LIN {X 0,Y 365.471,Z 705.441,A -85,B 0,C 180,E1 17669.142,E2 17669.142} C_VEL
LIN {X 0,Y 364.079,Z 703.275,A -85,B 0,C 180,E1 17668.635,E2 17668.635} C_VEL
LIN {X 0,Y 360.885,Z 700.431,A -85,B 0,C 180,E1 17667.516,E2 17667.516} C_VEL
LIN {X 0,Y 359.152,Z 697.27,A -85,B 0,C 180,E1 17666.808,E2 17666.808} C_VEL
LIN {X 0,Y 355.819,Z 694.962,A -85,B 0,C 180,E1 17665.553,E2 17665.553} C_VEL
LIN {X 0,Y 354.085,Z 691.734,A -85,B 0,C 180,E1 17664.704,E2 17664.704} C_VEL
LIN {X 0,Y 353.877,Z 690.724,A -85,B 0,C 180,E1 17664.135,E2 17664.135} C_VEL
LIN {X 0,Y 353.869,Z 690.629,A -85,B 0,C 180,E1 17659.992,E2 17659.992} C_VEL
LIN {X 0,Y 353.869,Z 690.628,A -85,B 0,C 180,E1 17655.739,E2 17655.739} C_VEL
LIN {X 0,Y 353.867,Z 690.628,A -85,B 0,C 180,E1 17651.573,E2 17651.573} C_VEL
LIN {X 0,Y 353.866,Z 690.63,A -85,B 0,C 180,E1 17647.374,E2 17647.374} C_VEL
LIN {X 0,Y 353.864,Z 690.635,A -85,B 0,C 180,E1 17643.078,E2 17643.078} C_VEL
LIN {X 0,Y 353.868,Z 690.646,A -85,B 0,C 180,E1 17638.867,E2 17638.867} C_VEL
LIN {X 0,Y 353.866,Z 690.656,A -85,B 0,C 180,E1 17634.65,E2 17634.65} C_VEL
LIN {X 0,Y 353.865,Z 690.656,A -85,B 0,C 180,E1 17630.404,E2 17630.404} C_VEL
LIN {X 0,Y 353.855,Z 690.604,A -85,B 0,C 180,E1 17626.103,E2 17626.103} C_VEL
LIN {X 0,Y 353.86,Z 690.613,A -85,B 0,C 180,E1 17622.062,E2 17622.062} C_VEL
LIN {X 0,Y 353.929,Z 691.075,A -85,B 0,C 180,E1 17620.528,E2 17620.528} C_VEL
LIN {X 0,Y 355.457,Z 694.509,A -85,B 0,C 180,E1 17619.242,E2 17619.242} C_VEL
LIN {X 0,Y 357.098,Z 696.566,A -85,B 0,C 180,E1 17618.31,E2 17618.31} C_VEL
LIN {X 0,Y 358.976,Z 700.206,A -85,B 0,C 180,E1 17617.049,E2 17617.049} C_VEL
LIN {X 0,Y 360.256,Z 702.129,A -85,B 0,C 180,E1 17616.328,E2 17616.328} C_VEL
LIN {X 0,Y 363.242,Z 707.517,A -85,B 0,C 180,E1 17614.571,E2 17614.571} C_VEL
LIN {X 0,Y 366.016,Z 712.562,A -85,B 0,C 180,E1 17613.034,E2 17613.034} C_VEL
LIN {X 0,Y 368.872,Z 717.077,A -85,B 0,C 180,E1 17611.859,E2 17611.859} C_VEL
LIN {X 0,Y 376.233,Z 727.791,A -85,B 0,C 180,E1 17609.541,E2 17609.541} C_VEL
LIN {X 0,Y 383.594,Z 738.851,A -85,B 0,C 180,E1 17607.436,E2 17607.436} C_VEL
LIN {X 0,Y 393.463,Z 754.803,A -85,B 0,C 180,E1 17604.86,E2 17604.86} C_VEL
LIN {X 0,Y 403.331,Z 772.096,A -85,B 0,C 180,E1 17602.512,E2 17602.512} C_VEL
LIN {X 0,Y 407.131,Z 779.707,A -85,B 0,C 180,E1 17601.643,E2 17601.643} C_VEL
LIN {X 0,Y 409.573,Z 806.484,A -85,B 0,C 180,E1 17600.521,E2 17600.521} C_VEL
LIN {X 0,Y 399.986,Z 1030.209,A -85,B 0,C 180,E1 17596.253,E2 17596.253} C_VEL
LIN {X 0,Y 398.316,Z 1052.933,A -85,B 0,C 180,E1 17595.707,E2 17595.707} C_VEL
LIN {X 0,Y 395.489,Z 1075.063,A -85,B 0,C 180,E1 17594.972,E2 17594.972} C_VEL
LIN {X 0,Y 391.945,Z 1096.948,A -85,B 0,C 180,E1 17593.997,E2 17593.997} C_VEL
LIN {X 0,Y 388.182,Z 1117.13,A -85,B 0,C 180,E1 17592.842,E2 17592.842} C_VEL
LIN {X 0,Y 383.951,Z 1137.009,A -85,B 0,C 180,E1 17591.409,E2 17591.409} C_VEL
LIN {X 0,Y 379.354,Z 1157.251,A -85,B 0,C 180,E1 17589.629,E2 17589.629} C_VEL
LIN {X 0,Y 374.862,Z 1176.045,A -85,B 0,C 180,E1 17587.646,E2 17587.646} C_VEL
LIN {X 0,Y 370.47,Z 1193.714,A -85,B 0,C 180,E1 17585.407,E2 17585.407} C_VEL
LIN {X 0,Y 366.21,Z 1211.069,A -85,B 0,C 180,E1 17582.807,E2 17582.807} C_VEL
LIN {X 0,Y 362.588,Z 1226.357,A -85,B 0,C 180,E1 17580.123,E2 17580.123} C_VEL
LIN {X 0,Y 359.384,Z 1240.715,A -85,B 0,C 180,E1 17577.146,E2 17577.146} C_VEL
LIN {X 0,Y 356.818,Z 1253.684,A -85,B 0,C 180,E1 17573.973,E2 17573.973} C_VEL
LIN {X 0,Y 354.911,Z 1265.27,A -85,B 0,C 180,E1 17570.618,E2 17570.618} C_VEL
LIN {X 0,Y 353.685,Z 1274.869,A -85,B 0,C 180,E1 17567.267,E2 17567.267} C_VEL
LIN {X 0,Y 353.03,Z 1282.602,A -85,B 0,C 180,E1 17563.93,E2 17563.93} C_VEL
LIN {X 0,Y 352.775,Z 1288.725,A -85,B 0,C 180,E1 17560.616,E2 17560.616} C_VEL
LIN {X 0,Y 352.788,Z 1293.069,A -85,B 0,C 180,E1 17557.327,E2 17557.327} C_VEL
LIN {X 0,Y 352.885,Z 1295.906,A -85,B 0,C 180,E1 17554.062,E2 17554.062} C_VEL
LIN {X 0,Y 352.961,Z 1297.035,A -85,B 0,C 180,E1 17550.974,E2 17550.974} C_VEL
LIN {X 0,Y 352.934,Z 1296.834,A -85,B 0,C 180,E1 17547.889,E2 17547.889} C_VEL
LIN {X 0,Y 352.868,Z 1295.066,A -85,B 0,C 180,E1 17544.798,E2 17544.798} C_VEL
LIN {X 0,Y 352.757,Z 1291.955,A -85,B 0,C 180,E1 17541.689,E2 17541.689} C_VEL
LIN {X 0,Y 352.832,Z 1287.019,A -85,B 0,C 180,E1 17538.393,E2 17538.393} C_VEL
LIN {X 0,Y 353.168,Z 1280.523,A -85,B 0,C 180,E1 17535.071,E2 17535.071} C_VEL
LIN {X 0,Y 353.99,Z 1272.151,A -85,B 0,C 180,E1 17531.729,E2 17531.729} C_VEL
LIN {X 0,Y 355.501,Z 1261.428,A -85,B 0,C 180,E1 17528.208,E2 17528.208} C_VEL
LIN {X 0,Y 357.626,Z 1249.512,A -85,B 0,C 180,E1 17524.937,E2 17524.937} C_VEL
LIN {X 0,Y 360.374,Z 1236.146,A -85,B 0,C 180,E1 17521.859,E2 17521.859} C_VEL
LIN {X 0,Y 363.819,Z 1220.969,A -85,B 0,C 180,E1 17518.892,E2 17518.892} C_VEL
LIN {X 0,Y 367.828,Z 1204.365,A -85,B 0,C 180,E1 17516.136,E2 17516.136} C_VEL
LIN {X 0,Y 372.136,Z 1187.097,A -85,B 0,C 180,E1 17513.71,E2 17513.71} C_VEL
LIN {X 0,Y 376.533,Z 1168.91,A -85,B 0,C 180,E1 17511.568,E2 17511.568} C_VEL
LIN {X 0,Y 381.215,Z 1149.171,A -85,B 0,C 180,E1 17509.623,E2 17509.623} C_VEL
LIN {X 0,Y 385.614,Z 1129.483,A -85,B 0,C 180,E1 17508.014,E2 17508.014} C_VEL
LIN {X 0,Y 389.739,Z 1108.779,A -85,B 0,C 180,E1 17506.655,E2 17506.655} C_VEL
LIN {X 0,Y 393.552,Z 1087.165,A -85,B 0,C 180,E1 17505.535,E2 17505.535} C_VEL
LIN {X 0,Y 396.831,Z 1065.352,A -85,B 0,C 180,E1 17504.682,E2 17504.682} C_VEL
LIN {X 0,Y 399.152,Z 1042.966,A -85,B 0,C 180,E1 17504.036,E2 17504.036} C_VEL
LIN {X 0,Y 400.876,Z 1008.481,A -85,B 0,C 180,E1 17503.333,E2 17503.333} C_VEL
LIN {X 0,Y 409.544,Z 804.991,A -85,B 0,C 180,E1 17499.449,E2 17499.449} C_VEL
LIN {X 0,Y 406.876,Z 778.87,A -85,B 0,C 180,E1 17498.307,E2 17498.307} C_VEL
LIN {X 0,Y 397.759,Z 762.191,A -85,B 0,C 180,E1 17496.208,E2 17496.208} C_VEL
LIN {X 0,Y 387.89,Z 745.698,A -85,B 0,C 180,E1 17493.744,E2 17493.744} C_VEL
LIN {X 0,Y 378.905,Z 731.771,A -85,B 0,C 180,E1 17491.277,E2 17491.277} C_VEL
LIN {X 0,Y 373.111,Z 723.252,A -85,B 0,C 180,E1 17489.543,E2 17489.543} C_VEL
LIN {X 0,Y 367.159,Z 714.598,A -85,B 0,C 180,E1 17487.577,E2 17487.577} C_VEL
LIN {X 0,Y 364.532,Z 709.935,A -85,B 0,C 180,E1 17486.206,E2 17486.206} C_VEL
LIN {X 0,Y 362.094,Z 705.482,A -85,B 0,C 180,E1 17484.817,E2 17484.817} C_VEL
LIN {X 0,Y 359.499,Z 700.812,A -85,B 0,C 180,E1 17483.262,E2 17483.262} C_VEL
LIN {X 0,Y 357.408,Z 697.484,A -85,B 0,C 180,E1 17482.016,E2 17482.016} C_VEL
LIN {X 0,Y 356.62,Z 695.787,A -85,B 0,C 180,E1 17481.44,E2 17481.44} C_VEL
LIN {X 0,Y 354.291,Z 692.379,A -85,B 0,C 180,E1 17479.992,E2 17479.992} C_VEL
LIN {X 0,Y 353.876,Z 690.761,A -85,B 0,C 180,E1 17479.323,E2 17479.323} C_VEL
LIN {X 0,Y 353.859,Z 690.626,A -85,B 0,C 180,E1 17475.067,E2 17475.067} C_VEL
LIN {X 0,Y 353.858,Z 690.634,A -85,B 0,C 180,E1 17470.748,E2 17470.748} C_VEL
LIN {X 0,Y 353.86,Z 690.635,A -85,B 0,C 180,E1 17466.489,E2 17466.489} C_VEL
LIN {X 0,Y 353.858,Z 690.63,A -85,B 0,C 180,E1 17462.267,E2 17462.267} C_VEL
LIN {X 0,Y 353.862,Z 690.627,A -85,B 0,C 180,E1 17458.219,E2 17458.219} C_VEL
LIN {X 0,Y 353.866,Z 690.63,A -85,B 0,C 180,E1 17453.999,E2 17453.999} C_VEL
LIN {X 0,Y 353.87,Z 690.639,A -85,B 0,C 180,E1 17449.911,E2 17449.911} C_VEL
LIN {X 0,Y 353.877,Z 690.644,A -85,B 0,C 180,E1 17445.603,E2 17445.603} C_VEL
LIN {X 0,Y 353.872,Z 690.647,A -85,B 0,C 180,E1 17441.38,E2 17441.38} C_VEL
LIN {X 0,Y 353.873,Z 690.644,A -85,B 0,C 180,E1 17437.084,E2 17437.084} C_VEL
LIN {X 0,Y 353.924,Z 691,A -85,B 0,C 180,E1 17435.456,E2 17435.456} C_VEL
LIN {X 0,Y 354.424,Z 692.729,A -85,B 0,C 180,E1 17434.91,E2 17434.91} C_VEL
LIN {X 0,Y 356.441,Z 695.597,A -85,B 0,C 180,E1 17434.049,E2 17434.049} C_VEL
LIN {X 0,Y 359.358,Z 697.669,A -85,B 0,C 180,E1 17432.963,E2 17432.963} C_VEL
LIN {X 0,Y 361.561,Z 701.257,A -85,B 0,C 180,E1 17432.092,E2 17432.092} C_VEL
LIN {X 0,Y 364.587,Z 703.891,A -85,B 0,C 180,E1 17431.05,E2 17431.05} C_VEL
LIN {X 0,Y 367.355,Z 707.815,A -85,B 0,C 180,E1 17430.081,E2 17430.081} C_VEL
LIN {X 0,Y 369.554,Z 709.947,A -85,B 0,C 180,E1 17429.381,E2 17429.381} C_VEL
LIN {X 0,Y 372.952,Z 714.372,A -85,B 0,C 180,E1 17428.3,E2 17428.3} C_VEL
LIN {X 0,Y 374.652,Z 716.424,A -85,B 0,C 180,E1 17427.786,E2 17427.786} C_VEL
LIN {X 0,Y 379.564,Z 722.657,A -85,B 0,C 180,E1 17426.354,E2 17426.354} C_VEL
LIN {X 0,Y 386.577,Z 731.681,A -85,B 0,C 180,E1 17424.458,E2 17424.458} C_VEL
LIN {X 0,Y 397.204,Z 746.475,A -85,B 0,C 180,E1 17421.831,E2 17421.831} C_VEL
LIN {X 0,Y 408.148,Z 762.945,A -85,B 0,C 180,E1 17419.381,E2 17419.381} C_VEL
LIN {X 0,Y 409.812,Z 765.853,A -85,B 0,C 180,E1 17419.02,E2 17419.02} C_VEL
LIN {X 0,Y 402.072,Z 938.592,A -85,B 0,C 180,E1 17415.686,E2 17415.686} C_VEL
LIN {X 0,Y 400.524,Z 960.749,A -85,B 0,C 180,E1 17415.004,E2 17415.004} C_VEL
LIN {X 0,Y 398.362,Z 981.552,A -85,B 0,C 180,E1 17414.123,E2 17414.123} C_VEL
LIN {X 0,Y 395.581,Z 1001.394,A -85,B 0,C 180,E1 17413.033,E2 17413.033} C_VEL
LIN {X 0,Y 392.215,Z 1020.769,A -85,B 0,C 180,E1 17411.708,E2 17411.708} C_VEL
LIN {X 0,Y 388.601,Z 1038.719,A -85,B 0,C 180,E1 17410.225,E2 17410.225} C_VEL
LIN {X 0,Y 384.411,Z 1056.584,A -85,B 0,C 180,E1 17408.435,E2 17408.435} C_VEL
LIN {X 0,Y 379.966,Z 1073.805,A -85,B 0,C 180,E1 17406.368,E2 17406.368} C_VEL
LIN {X 0,Y 375.604,Z 1089.572,A -85,B 0,C 180,E1 17404.118,E2 17404.118} C_VEL
LIN {X 0,Y 371.339,Z 1103.939,A -85,B 0,C 180,E1 17401.671,E2 17401.671} C_VEL
LIN {X 0,Y 367.297,Z 1117.2,A -85,B 0,C 180,E1 17398.982,E2 17398.982} C_VEL
LIN {X 0,Y 363.656,Z 1129.181,A -85,B 0,C 180,E1 17396.097,E2 17396.097} C_VEL
LIN {X 0,Y 360.477,Z 1139.749,A -85,B 0,C 180,E1 17393.022,E2 17393.022} C_VEL
LIN {X 0,Y 357.859,Z 1148.935,A -85,B 0,C 180,E1 17389.759,E2 17389.759} C_VEL
LIN {X 0,Y 355.866,Z 1156.767,A -85,B 0,C 180,E1 17386.317,E2 17386.317} C_VEL
LIN {X 0,Y 354.504,Z 1162.89,A -85,B 0,C 180,E1 17382.874,E2 17382.874} C_VEL
LIN {X 0,Y 353.689,Z 1167.41,A -85,B 0,C 180,E1 17379.388,E2 17379.388} C_VEL
LIN {X 0,Y 353.21,Z 1170.657,A -85,B 0,C 180,E1 17375.686,E2 17375.686} C_VEL
LIN {X 0,Y 353.051,Z 1172.217,A -85,B 0,C 180,E1 17372.4,E2 17372.4} C_VEL
LIN {X 0,Y 352.043,Z 1172.727,A -85,B 0,C 180,E1 17371.152,E2 17371.152} C_VEL
LIN {X 0,Y 347.31,Z 1173.512,A -85,B 0,C 180,E1 17368.703,E2 17368.703} C_VEL
LIN {X 0,Y 345.319,Z 1173.487,A -85,B 0,C 180,E1 17367.162,E2 17367.162} C_VEL
LIN {X 0,Y 345.197,Z 1173.339,A -85,B 0,C 180,E1 17366.699,E2 17366.699} C_VEL
LIN {X 0,Y 345.475,Z 1171.37,A -85,B 0,C 180,E1 17363.072,E2 17363.072} C_VEL
LIN {X 0,Y 346.007,Z 1168.136,A -85,B 0,C 180,E1 17359.679,E2 17359.679} C_VEL
LIN {X 0,Y 347.031,Z 1163.092,A -85,B 0,C 180,E1 17355.995,E2 17355.995} C_VEL
LIN {X 0,Y 348.637,Z 1156.696,A -85,B 0,C 180,E1 17352.475,E2 17352.475} C_VEL
LIN {X 0,Y 350.95,Z 1148.496,A -85,B 0,C 180,E1 17348.963,E2 17348.963} C_VEL
LIN {X 0,Y 353.886,Z 1138.82,A -85,B 0,C 180,E1 17345.639,E2 17345.639} C_VEL
LIN {X 0,Y 357.626,Z 1127.14,A -85,B 0,C 180,E1 17342.349,E2 17342.349} C_VEL
LIN {X 0,Y 361.695,Z 1114.634,A -85,B 0,C 180,E1 17339.428,E2 17339.428} C_VEL
LIN {X 0,Y 366.129,Z 1100.591,A -85,B 0,C 180,E1 17336.709,E2 17336.709} C_VEL
LIN {X 0,Y 370.63,Z 1085.712,A -85,B 0,C 180,E1 17334.294,E2 17334.294} C_VEL
LIN {X 0,Y 375.04,Z 1070.375,A -85,B 0,C 180,E1 17332.181,E2 17332.181} C_VEL
LIN {X 0,Y 379.54,Z 1053.085,A -85,B 0,C 180,E1 17330.198,E2 17330.198} C_VEL
LIN {X 0,Y 383.74,Z 1034.99,A -85,B 0,C 180,E1 17328.464,E2 17328.464} C_VEL
LIN {X 0,Y 387.565,Z 1016.262,A -85,B 0,C 180,E1 17326.973,E2 17326.973} C_VEL
LIN {X 0,Y 390.864,Z 996.564,A -85,B 0,C 180,E1 17325.707,E2 17325.707} C_VEL
LIN {X 0,Y 393.661,Z 975.449,A -85,B 0,C 180,E1 17324.633,E2 17324.633} C_VEL
LIN {X 0,Y 395.75,Z 954.159,A -85,B 0,C 180,E1 17323.812,E2 17323.812} C_VEL
LIN {X 0,Y 396.956,Z 933.715,A -85,B 0,C 180,E1 17323.253,E2 17323.253} C_VEL
LIN {X 0,Y 404.544,Z 769.328,A -85,B 0,C 180,E1 17320.063,E2 17320.063} C_VEL
LIN {X 0,Y 393.935,Z 753.113,A -85,B 0,C 180,E1 17317.62,E2 17317.62} C_VEL
LIN {X 0,Y 384.99,Z 740.534,A -85,B 0,C 180,E1 17315.367,E2 17315.367} C_VEL
LIN {X 0,Y 378.062,Z 731.268,A -85,B 0,C 180,E1 17313.465,E2 17313.465} C_VEL
LIN {X 0,Y 374.232,Z 726.376,A -85,B 0,C 180,E1 17312.346,E2 17312.346} C_VEL
LIN {X 0,Y 370.309,Z 721.384,A -85,B 0,C 180,E1 17311.136,E2 17311.136} C_VEL
LIN {X 0,Y 365.999,Z 715.983,A -85,B 0,C 180,E1 17309.725,E2 17309.725} C_VEL
LIN {X 0,Y 362.579,Z 711.859,A -85,B 0,C 180,E1 17308.539,E2 17308.539} C_VEL
LIN {X 0,Y 361.48,Z 710.424,A -85,B 0,C 180,E1 17308.139,E2 17308.139} C_VEL
LIN {X 0,Y 358.283,Z 707.187,A -85,B 0,C 180,E1 17306.968,E2 17306.968} C_VEL
LIN {X 0,Y 356.638,Z 704.578,A -85,B 0,C 180,E1 17306.293,E2 17306.293} C_VEL
LIN {X 0,Y 353.417,Z 701.9,A -85,B 0,C 180,E1 17305.021,E2 17305.021} C_VEL
LIN {X 0,Y 351.252,Z 698.256,A -85,B 0,C 180,E1 17304.02,E2 17304.02} C_VEL
LIN {X 0,Y 347.935,Z 696.011,A -85,B 0,C 180,E1 17302.559,E2 17302.559} C_VEL
LIN {X 0,Y 346.135,Z 692.717,A -85,B 0,C 180,E1 17301.522,E2 17301.522} C_VEL
LIN {X 0,Y 345.941,Z 691.687,A -85,B 0,C 180,E1 17300.824,E2 17300.824} C_VEL
LIN {X 0,Y 345.932,Z 691.618,A -85,B 0,C 180,E1 17296.455,E2 17296.455} C_VEL
LIN {X 0,Y 345.93,Z 691.62,A -85,B 0,C 180,E1 17292.181,E2 17292.181} C_VEL
LIN {X 0,Y 345.938,Z 691.621,A -85,B 0,C 180,E1 17287.808,E2 17287.808} C_VEL
LIN {X 0,Y 345.928,Z 691.629,A -85,B 0,C 180,E1 17283.48,E2 17283.48} C_VEL
LIN {X 0,Y 345.935,Z 691.64,A -85,B 0,C 180,E1 17279.172,E2 17279.172} C_VEL
LIN {X 0,Y 345.931,Z 691.647,A -85,B 0,C 180,E1 17274.86,E2 17274.86} C_VEL
LIN {X 0,Y 345.928,Z 691.638,A -85,B 0,C 180,E1 17270.685,E2 17270.685} C_VEL
LIN {X 0,Y 345.924,Z 691.587,A -85,B 0,C 180,E1 17266.46,E2 17266.46} C_VEL
LIN {X 0,Y 345.978,Z 691.985,A -85,B 0,C 180,E1 17263.32,E2 17263.32} C_VEL
LIN {X 0,Y 347.643,Z 695.648,A -85,B 0,C 180,E1 17261.73,E2 17261.73} C_VEL
LIN {X 0,Y 349.357,Z 697.89,A -85,B 0,C 180,E1 17260.611,E2 17260.611} C_VEL
LIN {X 0,Y 351.358,Z 701.541,A -85,B 0,C 180,E1 17259.163,E2 17259.163} C_VEL
LIN {X 0,Y 352.421,Z 703.029,A -85,B 0,C 180,E1 17258.52,E2 17258.52} C_VEL
LIN {X 0,Y 354.585,Z 706.924,A -85,B 0,C 180,E1 17257.1,E2 17257.1} C_VEL
LIN {X 0,Y 357.639,Z 711.946,A -85,B 0,C 180,E1 17255.471,E2 17255.471} C_VEL
LIN {X 0,Y 365.872,Z 723.456,A -85,B 0,C 180,E1 17252.45,E2 17252.45} C_VEL
LIN {X 0,Y 373.526,Z 734.859,A -85,B 0,C 180,E1 17249.963,E2 17249.963} C_VEL
LIN {X 0,Y 380.424,Z 745.435,A -85,B 0,C 180,E1 17247.933,E2 17247.933} C_VEL
LIN {X 0,Y 390.016,Z 761.232,A -85,B 0,C 180,E1 17245.356,E2 17245.356} C_VEL
LIN {X 0,Y 399.414,Z 777.97,A -85,B 0,C 180,E1 17243.051,E2 17243.051} C_VEL
LIN {X 0,Y 402.235,Z 783.755,A -85,B 0,C 180,E1 17242.381,E2 17242.381} C_VEL
LIN {X 0,Y 404.318,Z 807.97,A -85,B 0,C 180,E1 17241.354,E2 17241.354} C_VEL
LIN {X 0,Y 394.338,Z 1030.205,A -85,B 0,C 180,E1 17237.074,E2 17237.074} C_VEL
LIN {X 0,Y 392.557,Z 1052.868,A -85,B 0,C 180,E1 17236.516,E2 17236.516} C_VEL
LIN {X 0,Y 389.542,Z 1075.287,A -85,B 0,C 180,E1 17235.753,E2 17235.753} C_VEL
LIN {X 0,Y 385.961,Z 1096.296,A -85,B 0,C 180,E1 17234.798,E2 17234.798} C_VEL
LIN {X 0,Y 381.963,Z 1116.754,A -85,B 0,C 180,E1 17233.609,E2 17233.609} C_VEL
LIN {X 0,Y 377.446,Z 1137.037,A -85,B 0,C 180,E1 17232.122,E2 17232.122} C_VEL
LIN {X 0,Y 372.825,Z 1156.344,A -85,B 0,C 180,E1 17230.391,E2 17230.391} C_VEL
LIN {X 0,Y 368.084,Z 1175.208,A -85,B 0,C 180,E1 17228.365,E2 17228.365} C_VEL
LIN {X 0,Y 363.438,Z 1193.028,A -85,B 0,C 180,E1 17226.066,E2 17226.066} C_VEL
LIN {X 0,Y 359.03,Z 1210.026,A -85,B 0,C 180,E1 17223.462,E2 17223.462} C_VEL
LIN {X 0,Y 355.085,Z 1225.698,A -85,B 0,C 180,E1 17220.64,E2 17220.64} C_VEL
LIN {X 0,Y 351.612,Z 1240.558,A -85,B 0,C 180,E1 17217.475,E2 17217.475} C_VEL
LIN {X 0,Y 348.917,Z 1253.462,A -85,B 0,C 180,E1 17214.19,E2 17214.19} C_VEL
LIN {X 0,Y 346.958,Z 1264.821,A -85,B 0,C 180,E1 17210.76,E2 17210.76} C_VEL
LIN {X 0,Y 345.71,Z 1274.303,A -85,B 0,C 180,E1 17207.331,E2 17207.331} C_VEL
LIN {X 0,Y 345.065,Z 1281.866,A -85,B 0,C 180,E1 17203.907,E2 17203.907} C_VEL
LIN {X 0,Y 344.845,Z 1288.021,A -85,B 0,C 180,E1 17200.356,E2 17200.356} C_VEL
LIN {X 0,Y 344.882,Z 1292.027,A -85,B 0,C 180,E1 17197.161,E2 17197.161} C_VEL
LIN {X 0,Y 345.008,Z 1294.674,A -85,B 0,C 180,E1 17193.822,E2 17193.822} C_VEL
LIN {X 0,Y 345.08,Z 1295.669,A -85,B 0,C 180,E1 17190.83,E2 17190.83} C_VEL
LIN {X 0,Y 345.043,Z 1295.301,A -85,B 0,C 180,E1 17187.509,E2 17187.509} C_VEL
LIN {X 0,Y 344.951,Z 1293.532,A -85,B 0,C 180,E1 17184.511,E2 17184.511} C_VEL
LIN {X 0,Y 344.835,Z 1290.355,A -85,B 0,C 180,E1 17181.328,E2 17181.328} C_VEL
LIN {X 0,Y 344.914,Z 1285.3,A -85,B 0,C 180,E1 17177.953,E2 17177.953} C_VEL
LIN {X 0,Y 345.323,Z 1278.286,A -85,B 0,C 180,E1 17174.379,E2 17174.379} C_VEL
LIN {X 0,Y 346.187,Z 1270.233,A -85,B 0,C 180,E1 17171.127,E2 17171.127} C_VEL
LIN {X 0,Y 347.745,Z 1259.95,A -85,B 0,C 180,E1 17167.696,E2 17167.696} C_VEL
LIN {X 0,Y 349.949,Z 1248.388,A -85,B 0,C 180,E1 17164.442,E2 17164.442} C_VEL
LIN {X 0,Y 352.952,Z 1234.654,A -85,B 0,C 180,E1 17161.212,E2 17161.212} C_VEL
LIN {X 0,Y 356.618,Z 1219.477,A -85,B 0,C 180,E1 17158.191,E2 17158.191} C_VEL
LIN {X 0,Y 360.891,Z 1202.746,A -85,B 0,C 180,E1 17155.37,E2 17155.37} C_VEL
LIN {X 0,Y 365.456,Z 1185.367,A -85,B 0,C 180,E1 17152.897,E2 17152.897} C_VEL
LIN {X 0,Y 370.161,Z 1166.853,A -85,B 0,C 180,E1 17150.699,E2 17150.699} C_VEL
LIN {X 0,Y 375.092,Z 1147.001,A -85,B 0,C 180,E1 17148.738,E2 17148.738} C_VEL
LIN {X 0,Y 379.508,Z 1128.019,A -85,B 0,C 180,E1 17147.179,E2 17147.179} C_VEL
LIN {X 0,Y 383.778,Z 1107.455,A -85,B 0,C 180,E1 17145.821,E2 17145.821} C_VEL
LIN {X 0,Y 387.796,Z 1085.627,A -85,B 0,C 180,E1 17144.688,E2 17144.688} C_VEL
LIN {X 0,Y 391.182,Z 1063.831,A -85,B 0,C 180,E1 17143.835,E2 17143.835} C_VEL
LIN {X 0,Y 393.571,Z 1041.356,A -85,B 0,C 180,E1 17143.183,E2 17143.183} C_VEL
LIN {X 0,Y 395.395,Z 1006,A -85,B 0,C 180,E1 17142.458,E2 17142.458} C_VEL
LIN {X 0,Y 404.287,Z 806.378,A -85,B 0,C 180,E1 17138.613,E2 17138.613} C_VEL
LIN {X 0,Y 401.977,Z 782.959,A -85,B 0,C 180,E1 17137.568,E2 17137.568} C_VEL
LIN {X 0,Y 393.041,Z 766.442,A -85,B 0,C 180,E1 17135.428,E2 17135.428} C_VEL
LIN {X 0,Y 382.85,Z 749.242,A -85,B 0,C 180,E1 17132.769,E2 17132.769} C_VEL
LIN {X 0,Y 374.337,Z 736.079,A -85,B 0,C 180,E1 17130.319,E2 17130.319} C_VEL
LIN {X 0,Y 367.967,Z 726.664,A -85,B 0,C 180,E1 17128.304,E2 17128.304} C_VEL
LIN {X 0,Y 363.794,Z 720.659,A -85,B 0,C 180,E1 17126.879,E2 17126.879} C_VEL
LIN {X 0,Y 357.321,Z 711.598,A -85,B 0,C 180,E1 17124.465,E2 17124.465} C_VEL
LIN {X 0,Y 354.502,Z 706.829,A -85,B 0,C 180,E1 17122.906,E2 17122.906} C_VEL
LIN {X 0,Y 352.349,Z 702.839,A -85,B 0,C 180,E1 17121.473,E2 17121.473} C_VEL
LIN {X 0,Y 349.639,Z 698.685,A -85,B 0,C 180,E1 17119.721,E2 17119.721} C_VEL
LIN {X 0,Y 348.867,Z 696.937,A -85,B 0,C 180,E1 17119.07,E2 17119.07} C_VEL
LIN {X 0,Y 346.498,Z 693.756,A -85,B 0,C 180,E1 17117.463,E2 17117.463} C_VEL
LIN {X 0,Y 345.956,Z 691.853,A -85,B 0,C 180,E1 17116.626,E2 17116.626} C_VEL
LIN {X 0,Y 345.918,Z 691.588,A -85,B 0,C 180,E1 17112.52,E2 17112.52} C_VEL
LIN {X 0,Y 345.923,Z 691.621,A -85,B 0,C 180,E1 17108.309,E2 17108.309} C_VEL
LIN {X 0,Y 345.92,Z 691.629,A -85,B 0,C 180,E1 17104.144,E2 17104.144} C_VEL
LIN {X 0,Y 345.923,Z 691.637,A -85,B 0,C 180,E1 17099.834,E2 17099.834} C_VEL
LIN {X 0,Y 345.922,Z 691.647,A -85,B 0,C 180,E1 17095.524,E2 17095.524} C_VEL
LIN {X 0,Y 345.921,Z 691.641,A -85,B 0,C 180,E1 17091.299,E2 17091.299} C_VEL
LIN {X 0,Y 345.922,Z 691.634,A -85,B 0,C 180,E1 17086.97,E2 17086.97} C_VEL
LIN {X 0,Y 345.923,Z 691.629,A -85,B 0,C 180,E1 17082.679,E2 17082.679} C_VEL
LIN {X 0,Y 345.952,Z 691.793,A -85,B 0,C 180,E1 17078.821,E2 17078.821} C_VEL
LIN {X 0,Y 346.263,Z 693.135,A -85,B 0,C 180,E1 17078.175,E2 17078.175} C_VEL
LIN {X 0,Y 347.944,Z 696.018,A -85,B 0,C 180,E1 17077.272,E2 17077.272} C_VEL
LIN {X 0,Y 351.639,Z 698.72,A -85,B 0,C 180,E1 17075.651,E2 17075.651} C_VEL
LIN {X 0,Y 353.739,Z 702.299,A -85,B 0,C 180,E1 17074.69,E2 17074.69} C_VEL
LIN {X 0,Y 357.083,Z 705.131,A -85,B 0,C 180,E1 17073.384,E2 17073.384} C_VEL
LIN {X 0,Y 359.722,Z 708.944,A -85,B 0,C 180,E1 17072.342,E2 17072.342} C_VEL
LIN {X 0,Y 362.185,Z 711.201,A -85,B 0,C 180,E1 17071.472,E2 17071.472} C_VEL
LIN {X 0,Y 365.461,Z 715.501,A -85,B 0,C 180,E1 17070.317,E2 17070.317} C_VEL
LIN {X 0,Y 367.18,Z 717.401,A -85,B 0,C 180,E1 17069.75,E2 17069.75} C_VEL
LIN {X 0,Y 371.011,Z 722.061,A -85,B 0,C 180,E1 17068.523,E2 17068.523} C_VEL
LIN {X 0,Y 380.126,Z 733.931,A -85,B 0,C 180,E1 17065.835,E2 17065.835} C_VEL
LIN {X 0,Y 390.273,Z 747.832,A -85,B 0,C 180,E1 17063.166,E2 17063.166} C_VEL
LIN {X 0,Y 400.617,Z 763.242,A -85,B 0,C 180,E1 17060.705,E2 17060.705} C_VEL
LIN {X 0,Y 404.549,Z 769.661,A -85,B 0,C 180,E1 17059.821,E2 17059.821} C_VEL
LIN {X 0,Y 396.607,Z 939.648,A -85,B 0,C 180,E1 17056.512,E2 17056.512} C_VEL
LIN {X 0,Y 395.01,Z 961.899,A -85,B 0,C 180,E1 17055.823,E2 17055.823} C_VEL
LIN {X 0,Y 392.855,Z 982.158,A -85,B 0,C 180,E1 17054.965,E2 17054.965} C_VEL
LIN {X 0,Y 390.049,Z 1001.546,A -85,B 0,C 180,E1 17053.899,E2 17053.899} C_VEL
LIN {X 0,Y 386.561,Z 1021.196,A -85,B 0,C 180,E1 17052.56,E2 17052.56} C_VEL
LIN {X 0,Y 382.801,Z 1039.298,A -85,B 0,C 180,E1 17051.063,E2 17051.063} C_VEL
LIN {X 0,Y 378.512,Z 1056.971,A -85,B 0,C 180,E1 17049.287,E2 17049.287} C_VEL
LIN {X 0,Y 373.71,Z 1074.91,A -85,B 0,C 180,E1 17047.127,E2 17047.127} C_VEL
LIN {X 0,Y 369.147,Z 1090.744,A -85,B 0,C 180,E1 17044.845,E2 17044.845} C_VEL
LIN {X 0,Y 364.608,Z 1105.342,A -85,B 0,C 180,E1 17042.326,E2 17042.326} C_VEL
LIN {X 0,Y 360.362,Z 1118.605,A -85,B 0,C 180,E1 17039.595,E2 17039.595} C_VEL
LIN {X 0,Y 356.523,Z 1130.588,A -85,B 0,C 180,E1 17036.66,E2 17036.66} C_VEL
LIN {X 0,Y 353.07,Z 1141.461,A -85,B 0,C 180,E1 17033.431,E2 17033.431} C_VEL
LIN {X 0,Y 350.255,Z 1150.758,A -85,B 0,C 180,E1 17030.032,E2 17030.032} C_VEL
LIN {X 0,Y 348.069,Z 1158.805,A -85,B 0,C 180,E1 17026.35,E2 17026.35} C_VEL
LIN {X 0,Y 346.668,Z 1164.793,A -85,B 0,C 180,E1 17022.831,E2 17022.831} C_VEL
LIN {X 0,Y 345.828,Z 1169.118,A -85,B 0,C 180,E1 17019.317,E2 17019.317} C_VEL
LIN {X 0,Y 345.338,Z 1172.149,A -85,B 0,C 180,E1 17015.649,E2 17015.649} C_VEL
LIN {X 0,Y 345.169,Z 1173.714,A -85,B 0,C 180,E1 17012.158,E2 17012.158} C_VEL
LIN {X 0,Y 345.15,Z 1173.824,A -85,B 0,C 180,E1 17008.672,E2 17008.672} C_VEL
LIN {X 0,Y 345.197,Z 1173.339,A -85,B 0,C 180,E1 17006.699,E2 17006.699} C_VEL
LIN {X 0,Y 344.3,Z 1173.029,A -85,B 0,C 180,E1 17005.419,E2 17005.419} C_VEL
LIN {X 0,Y 338.432,Z 1171.92,A -85,B 0,C 180,E1 17001.889,E2 17001.889} C_VEL
LIN {X 0,Y 337.945,Z 1171.047,A -85,B 0,C 180,E1 17000.863,E2 17000.863} C_VEL
LIN {X 0,Y 338.794,Z 1166.769,A -85,B 0,C 180,E1 16997.213,E2 16997.213} C_VEL
LIN {X 0,Y 340.319,Z 1160.704,A -85,B 0,C 180,E1 16993.442,E2 16993.442} C_VEL
LIN {X 0,Y 342.476,Z 1153.233,A -85,B 0,C 180,E1 16989.849,E2 16989.849} C_VEL
LIN {X 0,Y 345.304,Z 1144.354,A -85,B 0,C 180,E1 16986.448,E2 16986.448} C_VEL
LIN {X 0,Y 348.721,Z 1134.068,A -85,B 0,C 180,E1 16983.247,E2 16983.247} C_VEL
LIN {X 0,Y 352.885,Z 1121.83,A -85,B 0,C 180,E1 16980.089,E2 16980.089} C_VEL
LIN {X 0,Y 357.264,Z 1108.919,A -85,B 0,C 180,E1 16977.308,E2 16977.308} C_VEL
LIN {X 0,Y 361.922,Z 1094.514,A -85,B 0,C 180,E1 16974.734,E2 16974.734} C_VEL
LIN {X 0,Y 366.923,Z 1078.185,A -85,B 0,C 180,E1 16972.285,E2 16972.285} C_VEL
LIN {X 0,Y 371.674,Z 1061.501,A -85,B 0,C 180,E1 16970.191,E2 16970.191} C_VEL
LIN {X 0,Y 376.142,Z 1043.857,A -85,B 0,C 180,E1 16968.354,E2 16968.354} C_VEL
LIN {X 0,Y 380.318,Z 1025.143,A -85,B 0,C 180,E1 16966.739,E2 16966.739} C_VEL
LIN {X 0,Y 383.874,Z 1006.668,A -85,B 0,C 180,E1 16965.418,E2 16965.418} C_VEL
LIN {X 0,Y 386.897,Z 986.887,A -85,B 0,C 180,E1 16964.289,E2 16964.289} C_VEL
LIN {X 0,Y 389.451,Z 965.005,A -85,B 0,C 180,E1 16963.315,E2 16963.315} C_VEL
LIN {X 0,Y 391.142,Z 943.712,A -85,B 0,C 180,E1 16962.617,E2 16962.617} C_VEL
LIN {X 0,Y 393.475,Z 894.086,A -85,B 0,C 180,E1 16961.592,E2 16961.592} C_VEL
LIN {X 0,Y 399.302,Z 773.086,A -85,B 0,C 180,E1 16959.227,E2 16959.227} C_VEL
LIN {X 0,Y 388.852,Z 757.058,A -85,B 0,C 180,E1 16956.715,E2 16956.715} C_VEL
LIN {X 0,Y 379.24,Z 743.486,A -85,B 0,C 180,E1 16954.165,E2 16954.165} C_VEL
LIN {X 0,Y 371.689,Z 733.528,A -85,B 0,C 180,E1 16951.956,E2 16951.956} C_VEL
LIN {X 0,Y 367.378,Z 728.068,A -85,B 0,C 180,E1 16950.594,E2 16950.594} C_VEL
LIN {X 0,Y 363.359,Z 722.964,A -85,B 0,C 180,E1 16949.238,E2 16949.238} C_VEL
LIN {X 0,Y 359.822,Z 718.436,A -85,B 0,C 180,E1 16947.964,E2 16947.964} C_VEL
LIN {X 0,Y 355.714,Z 713.936,A -85,B 0,C 180,E1 16946.412,E2 16946.412} C_VEL
LIN {X 0,Y 354.355,Z 711.94,A -85,B 0,C 180,E1 16945.846,E2 16945.846} C_VEL
LIN {X 0,Y 351.048,Z 708.817,A -85,B 0,C 180,E1 16944.483,E2 16944.483} C_VEL
LIN {X 0,Y 349.251,Z 705.805,A -85,B 0,C 180,E1 16943.629,E2 16943.629} C_VEL
LIN {X 0,Y 346.016,Z 703.383,A -85,B 0,C 180,E1 16942.154,E2 16942.154} C_VEL
LIN {X 0,Y 343.537,Z 699.321,A -85,B 0,C 180,E1 16940.799,E2 16940.799} C_VEL
LIN {X 0,Y 340.111,Z 697.121,A -85,B 0,C 180,E1 16938.957,E2 16938.957} C_VEL
LIN {X 0,Y 338.347,Z 694.193,A -85,B 0,C 180,E1 16937.765,E2 16937.765} C_VEL
LIN {X 0,Y 338.016,Z 692.83,A -85,B 0,C 180,E1 16936.968,E2 16936.968} C_VEL
LIN {X 0,Y 337.983,Z 692.618,A -85,B 0,C 180,E1 16932.819,E2 16932.819} C_VEL
LIN {X 0,Y 337.984,Z 692.624,A -85,B 0,C 180,E1 16928.506,E2 16928.506} C_VEL
LIN {X 0,Y 337.983,Z 692.635,A -85,B 0,C 180,E1 16924.242,E2 16924.242} C_VEL
LIN {X 0,Y 337.986,Z 692.632,A -85,B 0,C 180,E1 16919.831,E2 16919.831} C_VEL
LIN {X 0,Y 337.984,Z 692.624,A -85,B 0,C 180,E1 16915.419,E2 16915.419} C_VEL
LIN {X 0,Y 337.983,Z 692.617,A -85,B 0,C 180,E1 16911.132,E2 16911.132} C_VEL
LIN {X 0,Y 338.007,Z 692.769,A -85,B 0,C 180,E1 16906.834,E2 16906.834} C_VEL
LIN {X 0,Y 338.366,Z 694.239,A -85,B 0,C 180,E1 16905.978,E2 16905.978} C_VEL
LIN {X 0,Y 340.71,Z 697.74,A -85,B 0,C 180,E1 16903.987,E2 16903.987} C_VEL
LIN {X 0,Y 341.532,Z 698.997,A -85,B 0,C 180,E1 16903.328,E2 16903.328} C_VEL
LIN {X 0,Y 343.534,Z 702.617,A -85,B 0,C 180,E1 16901.68,E2 16901.68} C_VEL
LIN {X 0,Y 344.749,Z 704.274,A -85,B 0,C 180,E1 16900.869,E2 16900.869} C_VEL
LIN {X 0,Y 347.529,Z 708.457,A -85,B 0,C 180,E1 16899.364,E2 16899.364} C_VEL
LIN {X 0,Y 349.076,Z 710.636,A -85,B 0,C 180,E1 16898.625,E2 16898.625} C_VEL
LIN {X 0,Y 353.141,Z 716.095,A -85,B 0,C 180,E1 16896.825,E2 16896.825} C_VEL
LIN {X 0,Y 356.805,Z 721.318,A -85,B 0,C 180,E1 16895.321,E2 16895.321} C_VEL
LIN {X 0,Y 363.308,Z 730.531,A -85,B 0,C 180,E1 16892.905,E2 16892.905} C_VEL
LIN {X 0,Y 370.62,Z 741.58,A -85,B 0,C 180,E1 16890.461,E2 16890.461} C_VEL
LIN {X 0,Y 377.4,Z 752.207,A -85,B 0,C 180,E1 16888.406,E2 16888.406} C_VEL
LIN {X 0,Y 386.477,Z 767.433,A -85,B 0,C 180,E1 16885.892,E2 16885.892} C_VEL
LIN {X 0,Y 395.534,Z 783.843,A -85,B 0,C 180,E1 16883.601,E2 16883.601} C_VEL
LIN {X 0,Y 397.426,Z 787.914,A -85,B 0,C 180,E1 16883.131,E2 16883.131} C_VEL
LIN {X 0,Y 399.157,Z 809.331,A -85,B 0,C 180,E1 16882.212,E2 16882.212} C_VEL
LIN {X 0,Y 388.793,Z 1029.877,A -85,B 0,C 180,E1 16877.925,E2 16877.925} C_VEL
LIN {X 0,Y 386.923,Z 1052.241,A -85,B 0,C 180,E1 16877.362,E2 16877.362} C_VEL
LIN {X 0,Y 383.812,Z 1074.555,A -85,B 0,C 180,E1 16876.596,E2 16876.596} C_VEL
LIN {X 0,Y 380.065,Z 1095.582,A -85,B 0,C 180,E1 16875.628,E2 16875.628} C_VEL
LIN {X 0,Y 375.811,Z 1116.339,A -85,B 0,C 180,E1 16874.403,E2 16874.403} C_VEL
LIN {X 0,Y 371.264,Z 1135.957,A -85,B 0,C 180,E1 16872.948,E2 16872.948} C_VEL
LIN {X 0,Y 366.263,Z 1155.846,A -85,B 0,C 180,E1 16871.139,E2 16871.139} C_VEL
LIN {X 0,Y 361.189,Z 1175.01,A -85,B 0,C 180,E1 16869.032,E2 16869.032} C_VEL
LIN {X 0,Y 356.36,Z 1192.719,A -85,B 0,C 180,E1 16866.699,E2 16866.699} C_VEL
LIN {X 0,Y 351.746,Z 1209.526,A -85,B 0,C 180,E1 16864.053,E2 16864.053} C_VEL
LIN {X 0,Y 347.399,Z 1225.871,A -85,B 0,C 180,E1 16861.009,E2 16861.009} C_VEL
LIN {X 0,Y 343.928,Z 1240.004,A -85,B 0,C 180,E1 16857.899,E2 16857.899} C_VEL
LIN {X 0,Y 341.148,Z 1252.611,A -85,B 0,C 180,E1 16854.593,E2 16854.593} C_VEL
LIN {X 0,Y 339.089,Z 1263.862,A -85,B 0,C 180,E1 16851.083,E2 16851.083} C_VEL
LIN {X 0,Y 337.785,Z 1273.249,A -85,B 0,C 180,E1 16847.573,E2 16847.573} C_VEL
LIN {X 0,Y 337.121,Z 1280.751,A -85,B 0,C 180,E1 16844.075,E2 16844.075} C_VEL
LIN {X 0,Y 336.913,Z 1286.838,A -85,B 0,C 180,E1 16840.429,E2 16840.429} C_VEL
LIN {X 0,Y 336.973,Z 1290.802,A -85,B 0,C 180,E1 16837.159,E2 16837.159} C_VEL
LIN {X 0,Y 337.126,Z 1293.36,A -85,B 0,C 180,E1 16833.741,E2 16833.741} C_VEL
LIN {X 0,Y 337.201,Z 1294.279,A -85,B 0,C 180,E1 16830.849,E2 16830.849} C_VEL
LIN {X 0,Y 337.162,Z 1293.984,A -85,B 0,C 180,E1 16827.621,E2 16827.621} C_VEL
LIN {X 0,Y 337.042,Z 1292.129,A -85,B 0,C 180,E1 16824.382,E2 16824.382} C_VEL
LIN {X 0,Y 336.911,Z 1288.94,A -85,B 0,C 180,E1 16821.123,E2 16821.123} C_VEL
LIN {X 0,Y 336.981,Z 1283.868,A -85,B 0,C 180,E1 16817.665,E2 16817.665} C_VEL
LIN {X 0,Y 337.381,Z 1277.232,A -85,B 0,C 180,E1 16814.178,E2 16814.178} C_VEL
LIN {X 0,Y 338.344,Z 1268.768,A -85,B 0,C 180,E1 16810.673,E2 16810.673} C_VEL
LIN {X 0,Y 340.009,Z 1258.471,A -85,B 0,C 180,E1 16807.16,E2 16807.16} C_VEL
LIN {X 0,Y 342.37,Z 1246.9,A -85,B 0,C 180,E1 16803.834,E2 16803.834} C_VEL
LIN {X 0,Y 345.569,Z 1233.161,A -85,B 0,C 180,E1 16800.537,E2 16800.537} C_VEL
LIN {X 0,Y 349.458,Z 1217.982,A -85,B 0,C 180,E1 16797.46,E2 16797.46} C_VEL
LIN {X 0,Y 353.959,Z 1201.386,A -85,B 0,C 180,E1 16794.615,E2 16794.615} C_VEL
LIN {X 0,Y 358.615,Z 1184.466,A -85,B 0,C 180,E1 16792.167,E2 16792.167} C_VEL
LIN {X 0,Y 363.545,Z 1166.073,A -85,B 0,C 180,E1 16789.943,E2 16789.943} C_VEL
LIN {X 0,Y 368.711,Z 1146.229,A -85,B 0,C 180,E1 16787.95,E2 16787.95} C_VEL
LIN {X 0,Y 373.485,Z 1126.554,A -85,B 0,C 180,E1 16786.317,E2 16786.317} C_VEL
LIN {X 0,Y 378.049,Z 1105.473,A -85,B 0,C 180,E1 16784.923,E2 16784.923} C_VEL
LIN {X 0,Y 382.12,Z 1084.184,A -85,B 0,C 180,E1 16783.821,E2 16783.821} C_VEL
LIN {X 0,Y 385.64,Z 1062.15,A -85,B 0,C 180,E1 16782.958,E2 16782.958} C_VEL
LIN {X 0,Y 388.08,Z 1039.745,A -85,B 0,C 180,E1 16782.305,E2 16782.305} C_VEL
LIN {X 0,Y 390.014,Z 1003.402,A -85,B 0,C 180,E1 16781.556,E2 16781.556} C_VEL
LIN {X 0,Y 399.119,Z 807.757,A -85,B 0,C 180,E1 16777.755,E2 16777.755} C_VEL
LIN {X 0,Y 397.148,Z 787.017,A -85,B 0,C 180,E1 16776.811,E2 16776.811} C_VEL
LIN {X 0,Y 388.265,Z 770.543,A -85,B 0,C 180,E1 16774.599,E2 16774.599} C_VEL
LIN {X 0,Y 378.834,Z 754.557,A -85,B 0,C 180,E1 16772.039,E2 16772.039} C_VEL
LIN {X 0,Y 371.189,Z 742.473,A -85,B 0,C 180,E1 16769.756,E2 16769.756} C_VEL
LIN {X 0,Y 364.736,Z 732.81,A -85,B 0,C 180,E1 16767.643,E2 16767.643} C_VEL
LIN {X 0,Y 360.668,Z 726.823,A -85,B 0,C 180,E1 16766.198,E2 16766.198} C_VEL
LIN {X 0,Y 354.643,Z 718.255,A -85,B 0,C 180,E1 16763.864,E2 16763.864} C_VEL
LIN {X 0,Y 351.419,Z 713.813,A -85,B 0,C 180,E1 16762.499,E2 16762.499} C_VEL
LIN {X 0,Y 347.554,Z 708.503,A -85,B 0,C 180,E1 16760.723,E2 16760.723} C_VEL
LIN {X 0,Y 344.885,Z 704.609,A -85,B 0,C 180,E1 16759.299,E2 16759.299} C_VEL
LIN {X 0,Y 343.963,Z 703.07,A -85,B 0,C 180,E1 16758.648,E2 16758.648} C_VEL
LIN {X 0,Y 341.77,Z 699.679,A -85,B 0,C 180,E1 16757.011,E2 16757.011} C_VEL
LIN {X 0,Y 341.095,Z 698.101,A -85,B 0,C 180,E1 16756.344,E2 16756.344} C_VEL
LIN {X 0,Y 338.582,Z 694.775,A -85,B 0,C 180,E1 16754.362,E2 16754.362} C_VEL
LIN {X 0,Y 338.007,Z 692.756,A -85,B 0,C 180,E1 16753.298,E2 16753.298} C_VEL
LIN {X 0,Y 337.985,Z 692.62,A -85,B 0,C 180,E1 16749.02,E2 16749.02} C_VEL
LIN {X 0,Y 337.987,Z 692.628,A -85,B 0,C 180,E1 16744.751,E2 16744.751} C_VEL
LIN {X 0,Y 337.992,Z 692.635,A -85,B 0,C 180,E1 16740.339,E2 16740.339} C_VEL
LIN {X 0,Y 337.984,Z 692.63,A -85,B 0,C 180,E1 16735.928,E2 16735.928} C_VEL
LIN {X 0,Y 337.986,Z 692.619,A -85,B 0,C 180,E1 16731.665,E2 16731.665} C_VEL
LIN {X 0,Y 337.985,Z 692.614,A -85,B 0,C 180,E1 16727.354,E2 16727.354} C_VEL
LIN {X 0,Y 337.995,Z 692.683,A -85,B 0,C 180,E1 16723.031,E2 16723.031} C_VEL
LIN {X 0,Y 338.276,Z 693.965,A -85,B 0,C 180,E1 16722.097,E2 16722.097} C_VEL
LIN {X 0,Y 339.955,Z 696.953,A -85,B 0,C 180,E1 16720.945,E2 16720.945} C_VEL
LIN {X 0,Y 343.985,Z 699.88,A -85,B 0,C 180,E1 16718.784,E2 16718.784} C_VEL
LIN {X 0,Y 346.035,Z 703.409,A -85,B 0,C 180,E1 16717.668,E2 16717.668} C_VEL
LIN {X 0,Y 349.538,Z 706.198,A -85,B 0,C 180,E1 16716.079,E2 16716.079} C_VEL
LIN {X 0,Y 351.975,Z 709.97,A -85,B 0,C 180,E1 16714.959,E2 16714.959} C_VEL
LIN {X 0,Y 354.885,Z 712.562,A -85,B 0,C 180,E1 16713.792,E2 16713.792} C_VEL
LIN {X 0,Y 357.991,Z 716.703,A -85,B 0,C 180,E1 16712.558,E2 16712.558} C_VEL
LIN {X 0,Y 359.906,Z 718.61,A -85,B 0,C 180,E1 16711.863,E2 16711.863} C_VEL
LIN {X 0,Y 363.467,Z 723.073,A -85,B 0,C 180,E1 16710.591,E2 16710.591} C_VEL
LIN {X 0,Y 369.584,Z 730.883,A -85,B 0,C 180,E1 16708.57,E2 16708.57} C_VEL
LIN {X 0,Y 374.683,Z 737.49,A -85,B 0,C 180,E1 16707.017,E2 16707.017} C_VEL
LIN {X 0,Y 383.416,Z 749.239,A -85,B 0,C 180,E1 16704.579,E2 16704.579} C_VEL
LIN {X 0,Y 393.546,Z 764.174,A -85,B 0,C 180,E1 16702.014,E2 16702.014} C_VEL
LIN {X 0,Y 399.365,Z 773.486,A -85,B 0,C 180,E1 16700.642,E2 16700.642} C_VEL
LIN {X 0,Y 391.227,Z 940.702,A -85,B 0,C 180,E1 16697.361,E2 16697.361} C_VEL
LIN {X 0,Y 389.567,Z 963.179,A -85,B 0,C 180,E1 16696.659,E2 16696.659} C_VEL
LIN {X 0,Y 387.272,Z 983.893,A -85,B 0,C 180,E1 16695.771,E2 16695.771} C_VEL
LIN {X 0,Y 384.412,Z 1002.946,A -85,B 0,C 180,E1 16694.713,E2 16694.713} C_VEL
LIN {X 0,Y 380.682,Z 1023.144,A -85,B 0,C 180,E1 16693.319,E2 16693.319} C_VEL
LIN {X 0,Y 376.667,Z 1041.639,A -85,B 0,C 180,E1 16691.762,E2 16691.762} C_VEL
LIN {X 0,Y 372.174,Z 1059.38,A -85,B 0,C 180,E1 16689.946,E2 16689.946} C_VEL
LIN {X 0,Y 367.523,Z 1076.011,A -85,B 0,C 180,E1 16687.912,E2 16687.912} C_VEL
LIN {X 0,Y 362.687,Z 1092.1,A -85,B 0,C 180,E1 16685.568,E2 16685.568} C_VEL
LIN {X 0,Y 357.927,Z 1106.746,A -85,B 0,C 180,E1 16683.005,E2 16683.005} C_VEL
LIN {X 0,Y 353.469,Z 1120.011,A -85,B 0,C 180,E1 16680.231,E2 16680.231} C_VEL
LIN {X 0,Y 349.428,Z 1131.995,A -85,B 0,C 180,E1 16677.246,E2 16677.246} C_VEL
LIN {X 0,Y 345.795,Z 1142.805,A -85,B 0,C 180,E1 16673.977,E2 16673.977} C_VEL
LIN {X 0,Y 342.867,Z 1151.904,A -85,B 0,C 180,E1 16670.594,E2 16670.594} C_VEL
LIN {X 0,Y 340.53,Z 1159.894,A -85,B 0,C 180,E1 16666.898,E2 16666.898} C_VEL
LIN {X 0,Y 338.963,Z 1166.051,A -85,B 0,C 180,E1 16663.239,E2 16663.239} C_VEL
LIN {X 0,Y 338.018,Z 1170.516,A -85,B 0,C 180,E1 16659.535,E2 16659.535} C_VEL
LIN {X 0,Y 337.483,Z 1173.543,A -85,B 0,C 180,E1 16655.781,E2 16655.781} C_VEL
LIN {X 0,Y 337.294,Z 1175.105,A -85,B 0,C 180,E1 16652.208,E2 16652.208} C_VEL
LIN {X 0,Y 337.272,Z 1175.215,A -85,B 0,C 180,E1 16648.641,E2 16648.641} C_VEL
LIN {X 0,Y 337.43,Z 1173.999,A -85,B 0,C 180,E1 16644.9,E2 16644.9} C_VEL
LIN {X 0,Y 337.878,Z 1171.412,A -85,B 0,C 180,E1 16641.26,E2 16641.26} C_VEL
LIN {X 0,Y 337.945,Z 1171.047,A -85,B 0,C 180,E1 16640.863,E2 16640.863} C_VEL
LIN {X 0,Y 337.196,Z 1169.887,A -85,B 0,C 180,E1 16639.568,E2 16639.568} C_VEL
LIN {X 0,Y 332.084,Z 1166.864,A -85,B 0,C 180,E1 16636.07,E2 16636.07} C_VEL
LIN {X 0,Y 331.793,Z 1165.305,A -85,B 0,C 180,E1 16634.947,E2 16634.947} C_VEL
LIN {X 0,Y 333.8,Z 1158.408,A -85,B 0,C 180,E1 16631.126,E2 16631.126} C_VEL
LIN {X 0,Y 336.544,Z 1150.107,A -85,B 0,C 180,E1 16627.514,E2 16627.514} C_VEL
LIN {X 0,Y 340.012,Z 1140.05,A -85,B 0,C 180,E1 16624.014,E2 16624.014} C_VEL
LIN {X 0,Y 344.059,Z 1128.648,A -85,B 0,C 180,E1 16620.777,E2 16620.777} C_VEL
LIN {X 0,Y 348.643,Z 1115.851,A -85,B 0,C 180,E1 16617.764,E2 16617.764} C_VEL
LIN {X 0,Y 353.594,Z 1101.636,A -85,B 0,C 180,E1 16614.97,E2 16614.97} C_VEL
LIN {X 0,Y 358.62,Z 1086.238,A -85,B 0,C 180,E1 16612.47,E2 16612.47} C_VEL
LIN {X 0,Y 363.771,Z 1069.336,A -85,B 0,C 180,E1 16610.178,E2 16610.178} C_VEL
LIN {X 0,Y 368.441,Z 1052.58,A -85,B 0,C 180,E1 16608.27,E2 16608.27} C_VEL
LIN {X 0,Y 372.892,Z 1034.298,A -85,B 0,C 180,E1 16606.548,E2 16606.548} C_VEL
LIN {X 0,Y 377.013,Z 1014.654,A -85,B 0,C 180,E1 16605.029,E2 16605.029} C_VEL
LIN {X 0,Y 380.495,Z 994.754,A -85,B 0,C 180,E1 16603.783,E2 16603.783} C_VEL
LIN {X 0,Y 383.205,Z 974.605,A -85,B 0,C 180,E1 16602.793,E2 16602.793} C_VEL
LIN {X 0,Y 385.253,Z 953.337,A -85,B 0,C 180,E1 16602.005,E2 16602.005} C_VEL
LIN {X 0,Y 386.516,Z 931.802,A -85,B 0,C 180,E1 16601.438,E2 16601.438} C_VEL
LIN {X 0,Y 394.242,Z 777.025,A -85,B 0,C 180,E1 16598.392,E2 16598.392} C_VEL
LIN {X 0,Y 384.603,Z 762.197,A -85,B 0,C 180,E1 16595.983,E2 16595.983} C_VEL
LIN {X 0,Y 375.664,Z 749.464,A -85,B 0,C 180,E1 16593.524,E2 16593.524} C_VEL
LIN {X 0,Y 368.602,Z 740.027,A -85,B 0,C 180,E1 16591.387,E2 16591.387} C_VEL
LIN {X 0,Y 364.483,Z 734.728,A -85,B 0,C 180,E1 16590.043,E2 16590.043} C_VEL
LIN {X 0,Y 360.748,Z 729.919,A -85,B 0,C 180,E1 16588.743,E2 16588.743} C_VEL
LIN {X 0,Y 356.584,Z 724.719,A -85,B 0,C 180,E1 16587.197,E2 16587.197} C_VEL
LIN {X 0,Y 353.092,Z 720.538,A -85,B 0,C 180,E1 16585.81,E2 16585.81} C_VEL
LIN {X 0,Y 351.91,Z 719.11,A -85,B 0,C 180,E1 16585.316,E2 16585.316} C_VEL
LIN {X 0,Y 348.547,Z 715.475,A -85,B 0,C 180,E1 16583.859,E2 16583.859} C_VEL
LIN {X 0,Y 347.269,Z 713.33,A -85,B 0,C 180,E1 16583.232,E2 16583.232} C_VEL
LIN {X 0,Y 343.961,Z 710.566,A -85,B 0,C 180,E1 16581.665,E2 16581.665} C_VEL
LIN {X 0,Y 341.98,Z 707.076,A -85,B 0,C 180,E1 16580.54,E2 16580.54} C_VEL
LIN {X 0,Y 338.478,Z 704.673,A -85,B 0,C 180,E1 16578.605,E2 16578.605} C_VEL
LIN {X 0,Y 336.495,Z 701.35,A -85,B 0,C 180,E1 16577.242,E2 16577.242} C_VEL
LIN {X 0,Y 335.35,Z 700.202,A -85,B 0,C 180,E1 16576.454,E2 16576.454} C_VEL
LIN {X 0,Y 331.899,Z 697.81,A -85,B 0,C 180,E1 16573.857,E2 16573.857} C_VEL
LIN {X 0,Y 330.206,Z 694.446,A -85,B 0,C 180,E1 16571.883,E2 16571.883} C_VEL
LIN {X 0,Y 330.054,Z 693.648,A -85,B 0,C 180,E1 16570.296,E2 16570.296} C_VEL
LIN {X 0,Y 330.051,Z 693.594,A -85,B 0,C 180,E1 16565.912,E2 16565.912} C_VEL
LIN {X 0,Y 330.052,Z 693.592,A -85,B 0,C 180,E1 16561.476,E2 16561.476} C_VEL
LIN {X 0,Y 330.047,Z 693.592,A -85,B 0,C 180,E1 16557.222,E2 16557.222} C_VEL
LIN {X 0,Y 330.06,Z 693.591,A -85,B 0,C 180,E1 16552.866,E2 16552.866} C_VEL
LIN {X 0,Y 330.151,Z 694.229,A -85,B 0,C 180,E1 16550.764,E2 16550.764} C_VEL
LIN {X 0,Y 332.052,Z 697.957,A -85,B 0,C 180,E1 16548.449,E2 16548.449} C_VEL
LIN {X 0,Y 334.266,Z 700.171,A -85,B 0,C 180,E1 16546.684,E2 16546.684} C_VEL
LIN {X 0,Y 336.988,Z 704.311,A -85,B 0,C 180,E1 16544.689,E2 16544.689} C_VEL
LIN {X 0,Y 338.597,Z 706.192,A -85,B 0,C 180,E1 16543.664,E2 16543.664} C_VEL
LIN {X 0,Y 341.523,Z 710.226,A -85,B 0,C 180,E1 16541.921,E2 16541.921} C_VEL
LIN {X 0,Y 342.911,Z 712.04,A -85,B 0,C 180,E1 16541.16,E2 16541.16} C_VEL
LIN {X 0,Y 346.928,Z 717.773,A -85,B 0,C 180,E1 16539.106,E2 16539.106} C_VEL
LIN {X 0,Y 351.162,Z 723.628,A -85,B 0,C 180,E1 16537.174,E2 16537.174} C_VEL
LIN {X 0,Y 354.763,Z 728.908,A -85,B 0,C 180,E1 16535.658,E2 16535.658} C_VEL
LIN {X 0,Y 360.769,Z 737.59,A -85,B 0,C 180,E1 16533.367,E2 16533.367} C_VEL
LIN {X 0,Y 367.959,Z 748.635,A -85,B 0,C 180,E1 16530.896,E2 16530.896} C_VEL
LIN {X 0,Y 374.744,Z 759.539,A -85,B 0,C 180,E1 16528.783,E2 16528.783} C_VEL
LIN {X 0,Y 383.093,Z 773.85,A -85,B 0,C 180,E1 16526.406,E2 16526.406} C_VEL
LIN {X 0,Y 391.691,Z 789.715,A -85,B 0,C 180,E1 16524.161,E2 16524.161} C_VEL
LIN {X 0,Y 392.674,Z 791.991,A -85,B 0,C 180,E1 16523.904,E2 16523.904} C_VEL
LIN {X 0,Y 394.082,Z 810.809,A -85,B 0,C 180,E1 16523.089,E2 16523.089} C_VEL
LIN {X 0,Y 383.35,Z 1029.331,A -85,B 0,C 180,E1 16518.806,E2 16518.806} C_VEL
LIN {X 0,Y 381.339,Z 1051.874,A -85,B 0,C 180,E1 16518.225,E2 16518.225} C_VEL
LIN {X 0,Y 378.11,Z 1074.198,A -85,B 0,C 180,E1 16517.449,E2 16517.449} C_VEL
LIN {X 0,Y 374.277,Z 1094.737,A -85,B 0,C 180,E1 16516.492,E2 16516.492} C_VEL
LIN {X 0,Y 369.771,Z 1115.774,A -85,B 0,C 180,E1 16515.233,E2 16515.233} C_VEL
LIN {X 0,Y 365.029,Z 1135.432,A -85,B 0,C 180,E1 16513.757,E2 16513.757} C_VEL
LIN {X 0,Y 359.823,Z 1155.145,A -85,B 0,C 180,E1 16511.934,E2 16511.934} C_VEL
LIN {X 0,Y 354.344,Z 1174.813,A -85,B 0,C 180,E1 16509.725,E2 16509.725} C_VEL
LIN {X 0,Y 349.327,Z 1192.399,A -85,B 0,C 180,E1 16507.357,E2 16507.357} C_VEL
LIN {X 0,Y 344.499,Z 1209.026,A -85,B 0,C 180,E1 16504.67,E2 16504.67} C_VEL
LIN {X 0,Y 339.952,Z 1225.213,A -85,B 0,C 180,E1 16501.568,E2 16501.568} C_VEL
LIN {X 0,Y 336.263,Z 1239.417,A -85,B 0,C 180,E1 16498.342,E2 16498.342} C_VEL
LIN {X 0,Y 333.396,Z 1251.76,A -85,B 0,C 180,E1 16495.014,E2 16495.014} C_VEL
LIN {X 0,Y 331.231,Z 1262.903,A -85,B 0,C 180,E1 16491.422,E2 16491.422} C_VEL
LIN {X 0,Y 329.817,Z 1272.593,A -85,B 0,C 180,E1 16487.647,E2 16487.647} C_VEL
LIN {X 0,Y 329.156,Z 1279.997,A -85,B 0,C 180,E1 16484.064,E2 16484.064} C_VEL
LIN {X 0,Y 328.981,Z 1285.654,A -85,B 0,C 180,E1 16480.507,E2 16480.507} C_VEL
LIN {X 0,Y 329.064,Z 1289.578,A -85,B 0,C 180,E1 16477.156,E2 16477.156} C_VEL
LIN {X 0,Y 329.235,Z 1291.964,A -85,B 0,C 180,E1 16473.831,E2 16473.831} C_VEL
LIN {X 0,Y 329.323,Z 1292.888,A -85,B 0,C 180,E1 16470.87,E2 16470.87} C_VEL
LIN {X 0,Y 329.276,Z 1292.544,A -85,B 0,C 180,E1 16467.455,E2 16467.455} C_VEL
LIN {X 0,Y 329.135,Z 1290.727,A -85,B 0,C 180,E1 16464.247,E2 16464.247} C_VEL
LIN {X 0,Y 328.984,Z 1287.523,A -85,B 0,C 180,E1 16460.907,E2 16460.907} C_VEL
LIN {X 0,Y 329.046,Z 1282.433,A -85,B 0,C 180,E1 16457.363,E2 16457.363} C_VEL
LIN {X 0,Y 329.48,Z 1275.78,A -85,B 0,C 180,E1 16453.789,E2 16453.789} C_VEL
LIN {X 0,Y 330.525,Z 1267.271,A -85,B 0,C 180,E1 16450.184,E2 16450.184} C_VEL
LIN {X 0,Y 332.31,Z 1256.959,A -85,B 0,C 180,E1 16446.589,E2 16446.589} C_VEL
LIN {X 0,Y 334.829,Z 1245.411,A -85,B 0,C 180,E1 16443.199,E2 16443.199} C_VEL
LIN {X 0,Y 338.24,Z 1231.669,A -85,B 0,C 180,E1 16439.834,E2 16439.834} C_VEL
LIN {X 0,Y 342.358,Z 1216.487,A -85,B 0,C 180,E1 16436.699,E2 16436.699} C_VEL
LIN {X 0,Y 347.118,Z 1199.895,A -85,B 0,C 180,E1 16433.809,E2 16433.809} C_VEL
LIN {X 0,Y 352.19,Z 1182.393,A -85,B 0,C 180,E1 16431.246,E2 16431.246} C_VEL
LIN {X 0,Y 357.396,Z 1163.899,A -85,B 0,C 180,E1 16429.003,E2 16429.003} C_VEL
LIN {X 0,Y 362.85,Z 1143.687,A -85,B 0,C 180,E1 16426.972,E2 16426.972} C_VEL
LIN {X 0,Y 367.791,Z 1124.064,A -85,B 0,C 180,E1 16425.354,E2 16425.354} C_VEL
LIN {X 0,Y 372.456,Z 1103.393,A -85,B 0,C 180,E1 16423.993,E2 16423.993} C_VEL
LIN {X 0,Y 376.535,Z 1082.74,A -85,B 0,C 180,E1 16422.928,E2 16422.928} C_VEL
LIN {X 0,Y 380.11,Z 1061.103,A -85,B 0,C 180,E1 16422.076,E2 16422.076} C_VEL
LIN {X 0,Y 382.636,Z 1038.628,A -85,B 0,C 180,E1 16421.416,E2 16421.416} C_VEL
LIN {X 0,Y 384.59,Z 1003.833,A -85,B 0,C 180,E1 16420.688,E2 16420.688} C_VEL
LIN {X 0,Y 394.038,Z 809.056,A -85,B 0,C 180,E1 16416.872,E2 16416.872} C_VEL
LIN {X 0,Y 392.388,Z 791.109,A -85,B 0,C 180,E1 16416.036,E2 16416.036} C_VEL
LIN {X 0,Y 383.681,Z 774.978,A -85,B 0,C 180,E1 16413.783,E2 16413.783} C_VEL
LIN {X 0,Y 375.462,Z 760.754,A -85,B 0,C 180,E1 16411.463,E2 16411.463} C_VEL
LIN {X 0,Y 368.187,Z 749.028,A -85,B 0,C 180,E1 16409.218,E2 16409.218} C_VEL
LIN {X 0,Y 361.66,Z 739.078,A -85,B 0,C 180,E1 16407.006,E2 16407.006} C_VEL
LIN {X 0,Y 356.737,Z 731.631,A -85,B 0,C 180,E1 16405.171,E2 16405.171} C_VEL
LIN {X 0,Y 349.739,Z 721.546,A -85,B 0,C 180,E1 16402.259,E2 16402.259} C_VEL
LIN {X 0,Y 346.325,Z 716.76,A -85,B 0,C 180,E1 16400.667,E2 16400.667} C_VEL
LIN {X 0,Y 342.625,Z 711.591,A -85,B 0,C 180,E1 16398.767,E2 16398.767} C_VEL
LIN {X 0,Y 338.628,Z 706.335,A -85,B 0,C 180,E1 16396.466,E2 16396.466} C_VEL
LIN {X 0,Y 337.333,Z 704.692,A -85,B 0,C 180,E1 16395.648,E2 16395.648} C_VEL
LIN {X 0,Y 334.509,Z 700.759,A -85,B 0,C 180,E1 16393.658,E2 16393.658} C_VEL
LIN {X 0,Y 333.665,Z 699.392,A -85,B 0,C 180,E1 16392.988,E2 16392.988} C_VEL
LIN {X 0,Y 330.893,Z 696.319,A -85,B 0,C 180,E1 16390.621,E2 16390.621} C_VEL
LIN {X 0,Y 330.145,Z 694.209,A -85,B 0,C 180,E1 16389.412,E2 16389.412} C_VEL
LIN {X 0,Y 330.051,Z 693.592,A -85,B 0,C 180,E1 16387.31,E2 16387.31} C_VEL
LIN {X 0,Y 330.046,Z 693.592,A -85,B 0,C 180,E1 16382.952,E2 16382.952} C_VEL
LIN {X 0,Y 330.051,Z 693.593,A -85,B 0,C 180,E1 16378.611,E2 16378.611} C_VEL
LIN {X 0,Y 330.053,Z 693.596,A -85,B 0,C 180,E1 16374.262,E2 16374.262} C_VEL
LIN {X 0,Y 330.054,Z 693.621,A -85,B 0,C 180,E1 16369.88,E2 16369.88} C_VEL
LIN {X 0,Y 330.14,Z 694.144,A -85,B 0,C 180,E1 16368.115,E2 16368.115} C_VEL
LIN {X 0,Y 330.664,Z 695.85,A -85,B 0,C 180,E1 16367.07,E2 16367.07} C_VEL
LIN {X 0,Y 332.731,Z 698.645,A -85,B 0,C 180,E1 16365.201,E2 16365.201} C_VEL
LIN {X 0,Y 336.289,Z 700.934,A -85,B 0,C 180,E1 16362.703,E2 16362.703} C_VEL
LIN {X 0,Y 338.321,Z 704.503,A -85,B 0,C 180,E1 16361.297,E2 16361.297} C_VEL
LIN {X 0,Y 342.109,Z 707.406,A -85,B 0,C 180,E1 16359.2,E2 16359.2} C_VEL
LIN {X 0,Y 344.442,Z 711.137,A -85,B 0,C 180,E1 16357.919,E2 16357.919} C_VEL
LIN {X 0,Y 347.543,Z 713.75,A -85,B 0,C 180,E1 16356.473,E2 16356.473} C_VEL
LIN {X 0,Y 350.413,Z 717.822,A -85,B 0,C 180,E1 16355.148,E2 16355.148} C_VEL
LIN {X 0,Y 352.799,Z 720.082,A -85,B 0,C 180,E1 16354.167,E2 16354.167} C_VEL
LIN {X 0,Y 356.07,Z 724.26,A -85,B 0,C 180,E1 16352.851,E2 16352.851} C_VEL
LIN {X 0,Y 357.743,Z 726.125,A -85,B 0,C 180,E1 16352.221,E2 16352.221} C_VEL
LIN {X 0,Y 362.497,Z 732.149,A -85,B 0,C 180,E1 16350.505,E2 16350.505} C_VEL
LIN {X 0,Y 367.297,Z 738.384,A -85,B 0,C 180,E1 16348.899,E2 16348.899} C_VEL
LIN {X 0,Y 373.959,Z 747.087,A -85,B 0,C 180,E1 16346.854,E2 16346.854} C_VEL
LIN {X 0,Y 383.916,Z 761.22,A -85,B 0,C 180,E1 16344.081,E2 16344.081} C_VEL
LIN {X 0,Y 393.927,Z 776.577,A -85,B 0,C 180,E1 16341.571,E2 16341.571} C_VEL
LIN {X 0,Y 394.247,Z 777.657,A -85,B 0,C 180,E1 16341.478,E2 16341.478} C_VEL
LIN {X 0,Y 385.937,Z 941.742,A -85,B 0,C 180,E1 16338.233,E2 16338.233} C_VEL
LIN {X 0,Y 384.222,Z 964.33,A -85,B 0,C 180,E1 16337.524,E2 16337.524} C_VEL
LIN {X 0,Y 381.904,Z 984.717,A -85,B 0,C 180,E1 16336.648,E2 16336.648} C_VEL
LIN {X 0,Y 378.855,Z 1004.344,A -85,B 0,C 180,E1 16335.551,E2 16335.551} C_VEL
LIN {X 0,Y 375.114,Z 1023.952,A -85,B 0,C 180,E1 16334.191,E2 16334.191} C_VEL
LIN {X 0,Y 370.949,Z 1042.542,A -85,B 0,C 180,E1 16332.621,E2 16332.621} C_VEL
LIN {X 0,Y 366.347,Z 1060.075,A -85,B 0,C 180,E1 16330.817,E2 16330.817} C_VEL
LIN {X 0,Y 361.187,Z 1077.829,A -85,B 0,C 180,E1 16328.625,E2 16328.625} C_VEL
LIN {X 0,Y 356.272,Z 1093.501,A -85,B 0,C 180,E1 16326.309,E2 16326.309} C_VEL
LIN {X 0,Y 351.3,Z 1108.149,A -85,B 0,C 180,E1 16323.71,E2 16323.71} C_VEL
LIN {X 0,Y 346.623,Z 1121.417,A -85,B 0,C 180,E1 16320.893,E2 16320.893} C_VEL
LIN {X 0,Y 342.37,Z 1133.402,A -85,B 0,C 180,E1 16317.856,E2 16317.856} C_VEL
LIN {X 0,Y 338.552,Z 1144.149,A -85,B 0,C 180,E1 16314.545,E2 16314.545} C_VEL
LIN {X 0,Y 335.442,Z 1153.252,A -85,B 0,C 180,E1 16311.098,E2 16311.098} C_VEL
LIN {X 0,Y 332.921,Z 1161.3,A -85,B 0,C 180,E1 16307.296,E2 16307.296} C_VEL
LIN {X 0,Y 331.256,Z 1167.376,A -85,B 0,C 180,E1 16303.609,E2 16303.609} C_VEL
LIN {X 0,Y 330.213,Z 1171.914,A -85,B 0,C 180,E1 16299.762,E2 16299.762} C_VEL
LIN {X 0,Y 329.63,Z 1174.936,A -85,B 0,C 180,E1 16295.919,E2 16295.919} C_VEL
LIN {X 0,Y 329.42,Z 1176.496,A -85,B 0,C 180,E1 16292.261,E2 16292.261} C_VEL
LIN {X 0,Y 329.394,Z 1176.605,A -85,B 0,C 180,E1 16288.609,E2 16288.609} C_VEL
LIN {X 0,Y 329.567,Z 1175.392,A -85,B 0,C 180,E1 16284.778,E2 16284.778} C_VEL
LIN {X 0,Y 330.047,Z 1172.856,A -85,B 0,C 180,E1 16281.112,E2 16281.112} C_VEL
LIN {X 0,Y 330.892,Z 1168.831,A -85,B 0,C 180,E1 16277.426,E2 16277.426} C_VEL
LIN {X 0,Y 331.793,Z 1165.305,A -85,B 0,C 180,E1 16274.947,E2 16274.947} C_VEL
LIN {X 0,Y 331.417,Z 1163.486,A -85,B 0,C 180,E1 16273.644,E2 16273.644} C_VEL
LIN {X 0,Y 327.456,Z 1158.728,A -85,B 0,C 180,E1 16270.205,E2 16270.205} C_VEL
LIN {X 0,Y 327.476,Z 1156.33,A -85,B 0,C 180,E1 16269.014,E2 16269.014} C_VEL
LIN {X 0,Y 330.757,Z 1147.162,A -85,B 0,C 180,E1 16265.345,E2 16265.345} C_VEL
LIN {X 0,Y 334.569,Z 1136.876,A -85,B 0,C 180,E1 16262.019,E2 16262.019} C_VEL
LIN {X 0,Y 339.199,Z 1124.604,A -85,B 0,C 180,E1 16258.742,E2 16258.742} C_VEL
LIN {X 0,Y 344.007,Z 1111.715,A -85,B 0,C 180,E1 16255.879,E2 16255.879} C_VEL
LIN {X 0,Y 349.101,Z 1097.304,A -85,B 0,C 180,E1 16253.232,E2 16253.232} C_VEL
LIN {X 0,Y 354.536,Z 1080.97,A -85,B 0,C 180,E1 16250.72,E2 16250.72} C_VEL
LIN {X 0,Y 359.681,Z 1064.279,A -85,B 0,C 180,E1 16248.579,E2 16248.579} C_VEL
LIN {X 0,Y 364.505,Z 1046.63,A -85,B 0,C 180,E1 16246.706,E2 16246.706} C_VEL
LIN {X 0,Y 368.917,Z 1028.273,A -85,B 0,C 180,E1 16245.09,E2 16245.09} C_VEL
LIN {X 0,Y 372.814,Z 1009.433,A -85,B 0,C 180,E1 16243.718,E2 16243.718} C_VEL
LIN {X 0,Y 376.06,Z 989.649,A -85,B 0,C 180,E1 16242.569,E2 16242.569} C_VEL
LIN {X 0,Y 378.799,Z 967.786,A -85,B 0,C 180,E1 16241.579,E2 16241.579} C_VEL
LIN {X 0,Y 380.613,Z 946.593,A -85,B 0,C 180,E1 16240.87,E2 16240.87} C_VEL
LIN {X 0,Y 382.907,Z 901.231,A -85,B 0,C 180,E1 16239.905,E2 16239.905} C_VEL
LIN {X 0,Y 389.222,Z 780.986,A -85,B 0,C 180,E1 16237.528,E2 16237.528} C_VEL
LIN {X 0,Y 379.696,Z 766.198,A -85,B 0,C 180,E1 16235.034,E2 16235.034} C_VEL
LIN {X 0,Y 369.987,Z 752.351,A -85,B 0,C 180,E1 16232.212,E2 16232.212} C_VEL
LIN {X 0,Y 362.151,Z 742.002,A -85,B 0,C 180,E1 16229.663,E2 16229.663} C_VEL
LIN {X 0,Y 358.165,Z 736.862,A -85,B 0,C 180,E1 16228.241,E2 16228.241} C_VEL
LIN {X 0,Y 354.275,Z 731.918,A -85,B 0,C 180,E1 16226.754,E2 16226.754} C_VEL
LIN {X 0,Y 350.681,Z 727.425,A -85,B 0,C 180,E1 16225.275,E2 16225.275} C_VEL
LIN {X 0,Y 346.409,Z 722.625,A -85,B 0,C 180,E1 16223.383,E2 16223.383} C_VEL
LIN {X 0,Y 345.134,Z 720.731,A -85,B 0,C 180,E1 16222.753,E2 16222.753} C_VEL
LIN {X 0,Y 341.785,Z 717.538,A -85,B 0,C 180,E1 16221.09,E2 16221.09} C_VEL
LIN {X 0,Y 340.124,Z 714.66,A -85,B 0,C 180,E1 16220.118,E2 16220.118} C_VEL
LIN {X 0,Y 336.731,Z 712.073,A -85,B 0,C 180,E1 16218.167,E2 16218.167} C_VEL
LIN {X 0,Y 334.704,Z 708.503,A -85,B 0,C 180,E1 16216.71,E2 16216.71} C_VEL
LIN {X 0,Y 330.455,Z 705.393,A -85,B 0,C 180,E1 16213.473,E2 16213.473} C_VEL
LIN {X 0,Y 328.379,Z 701.767,A -85,B 0,C 180,E1 16211.237,E2 16211.237} C_VEL
LIN {X 0,Y 323.877,Z 698.691,A -85,B 0,C 180,E1 16202.832,E2 16202.832} C_VEL
LIN {X 0,Y 324.064,Z 698.913,A -85,B 0,C 180,E1 16198.586,E2 16198.586} C_VEL
LIN {X 0,Y 328.498,Z 701.876,A -85,B 0,C 180,E1 16191.07,E2 16191.07} C_VEL
LIN {X 0,Y 330.979,Z 705.962,A -85,B 0,C 180,E1 16188.5,E2 16188.5} C_VEL
LIN {X 0,Y 332.791,Z 707.838,A -85,B 0,C 180,E1 16187.022,E2 16187.022} C_VEL
LIN {X 0,Y 335.513,Z 711.994,A -85,B 0,C 180,E1 16184.974,E2 16184.974} C_VEL
LIN {X 0,Y 336.948,Z 713.773,A -85,B 0,C 180,E1 16184.03,E2 16184.03} C_VEL
LIN {X 0,Y 340.115,Z 718.055,A -85,B 0,C 180,E1 16182.109,E2 16182.109} C_VEL
LIN {X 0,Y 344.958,Z 725.172,A -85,B 0,C 180,E1 16179.513,E2 16179.513} C_VEL
LIN {X 0,Y 349.282,Z 731.281,A -85,B 0,C 180,E1 16177.489,E2 16177.489} C_VEL
LIN {X 0,Y 356.026,Z 741.224,A -85,B 0,C 180,E1 16174.686,E2 16174.686} C_VEL
LIN {X 0,Y 363.95,Z 753.481,A -85,B 0,C 180,E1 16171.802,E2 16171.802} C_VEL
LIN {X 0,Y 371.097,Z 765.157,A -85,B 0,C 180,E1 16169.478,E2 16169.478} C_VEL
LIN {X 0,Y 379.563,Z 779.937,A -85,B 0,C 180,E1 16166.979,E2 16166.979} C_VEL
LIN {X 0,Y 387.949,Z 795.707,A -85,B 0,C 180,E1 16164.716,E2 16164.716} C_VEL
LIN {X 0,Y 389.112,Z 812.075,A -85,B 0,C 180,E1 16163.993,E2 16163.993} C_VEL
LIN {X 0,Y 378.002,Z 1028.786,A -85,B 0,C 180,E1 16159.712,E2 16159.712} C_VEL
LIN {X 0,Y 375.788,Z 1051.947,A -85,B 0,C 180,E1 16159.099,E2 16159.099} C_VEL
LIN {X 0,Y 372.472,Z 1073.96,A -85,B 0,C 180,E1 16158.323,E2 16158.323} C_VEL
LIN {X 0,Y 368.431,Z 1094.613,A -85,B 0,C 180,E1 16157.343,E2 16157.343} C_VEL
LIN {X 0,Y 363.737,Z 1115.511,A -85,B 0,C 180,E1 16156.069,E2 16156.069} C_VEL
LIN {X 0,Y 358.871,Z 1134.906,A -85,B 0,C 180,E1 16154.594,E2 16154.594} C_VEL
LIN {X 0,Y 353.461,Z 1154.445,A -85,B 0,C 180,E1 16152.756,E2 16152.756} C_VEL
LIN {X 0,Y 347.746,Z 1173.976,A -85,B 0,C 180,E1 16150.526,E2 16150.526} C_VEL
LIN {X 0,Y 342.511,Z 1191.463,A -85,B 0,C 180,E1 16148.126,E2 16148.126} C_VEL
LIN {X 0,Y 337.293,Z 1208.525,A -85,B 0,C 180,E1 16145.312,E2 16145.312} C_VEL
LIN {X 0,Y 332.784,Z 1223.724,A -85,B 0,C 180,E1 16142.33,E2 16142.33} C_VEL
LIN {X 0,Y 328.931,Z 1237.695,A -85,B 0,C 180,E1 16139.1,E2 16139.1} C_VEL
LIN {X 0,Y 325.663,Z 1250.909,A -85,B 0,C 180,E1 16135.456,E2 16135.456} C_VEL
LIN {X 0,Y 323.383,Z 1261.943,A -85,B 0,C 180,E1 16131.778,E2 16131.778} C_VEL
LIN {X 0,Y 321.899,Z 1271.536,A -85,B 0,C 180,E1 16127.908,E2 16127.908} C_VEL
LIN {X 0,Y 321.208,Z 1278.899,A -85,B 0,C 180,E1 16124.235,E2 16124.235} C_VEL
LIN {X 0,Y 321.048,Z 1284.47,A -85,B 0,C 180,E1 16120.588,E2 16120.588} C_VEL
LIN {X 0,Y 321.164,Z 1288.516,A -85,B 0,C 180,E1 16116.974,E2 16116.974} C_VEL
LIN {X 0,Y 321.361,Z 1290.731,A -85,B 0,C 180,E1 16113.568,E2 16113.568} C_VEL
LIN {X 0,Y 321.445,Z 1291.572,A -85,B 0,C 180,E1 16110.356,E2 16110.356} C_VEL
LIN {X 0,Y 321.386,Z 1290.968,A -85,B 0,C 180,E1 16106.968,E2 16106.968} C_VEL
LIN {X 0,Y 321.224,Z 1289.191,A -85,B 0,C 180,E1 16103.925,E2 16103.925} C_VEL
LIN {X 0,Y 321.056,Z 1285.654,A -85,B 0,C 180,E1 16100.319,E2 16100.319} C_VEL
LIN {X 0,Y 321.122,Z 1280.703,A -85,B 0,C 180,E1 16096.863,E2 16096.863} C_VEL
LIN {X 0,Y 321.683,Z 1273.532,A -85,B 0,C 180,E1 16093.013,E2 16093.013} C_VEL
LIN {X 0,Y 322.902,Z 1264.726,A -85,B 0,C 180,E1 16089.249,E2 16089.249} C_VEL
LIN {X 0,Y 324.871,Z 1254.367,A -85,B 0,C 180,E1 16085.643,E2 16085.643} C_VEL
LIN {X 0,Y 327.827,Z 1241.839,A -85,B 0,C 180,E1 16081.987,E2 16081.987} C_VEL
LIN {X 0,Y 331.406,Z 1228.653,A -85,B 0,C 180,E1 16078.741,E2 16078.741} C_VEL
LIN {X 0,Y 335.61,Z 1214.089,A -85,B 0,C 180,E1 16075.733,E2 16075.733} C_VEL
LIN {X 0,Y 340.823,Z 1196.788,A -85,B 0,C 180,E1 16072.715,E2 16072.715} C_VEL
LIN {X 0,Y 346.002,Z 1179.846,A -85,B 0,C 180,E1 16070.234,E2 16070.234} C_VEL
LIN {X 0,Y 351.352,Z 1161.725,A -85,B 0,C 180,E1 16068.031,E2 16068.031} C_VEL
LIN {X 0,Y 356.802,Z 1142.298,A -85,B 0,C 180,E1 16066.069,E2 16066.069} C_VEL
LIN {X 0,Y 362.067,Z 1122.23,A -85,B 0,C 180,E1 16064.411,E2 16064.411} C_VEL
LIN {X 0,Y 366.824,Z 1101.944,A -85,B 0,C 180,E1 16063.074,E2 16063.074} C_VEL
LIN {X 0,Y 370.943,Z 1081.851,A -85,B 0,C 180,E1 16062.034,E2 16062.034} C_VEL
LIN {X 0,Y 374.64,Z 1060.304,A -85,B 0,C 180,E1 16061.176,E2 16061.176} C_VEL
LIN {X 0,Y 377.269,Z 1037.675,A -85,B 0,C 180,E1 16060.505,E2 16060.505} C_VEL
LIN {X 0,Y 379.233,Z 1004.749,A -85,B 0,C 180,E1 16059.806,E2 16059.806} C_VEL
LIN {X 0,Y 389.073,Z 810.592,A -85,B 0,C 180,E1 16055.976,E2 16055.976} C_VEL
LIN {X 0,Y 387.752,Z 795.431,A -85,B 0,C 180,E1 16055.259,E2 16055.259} C_VEL
LIN {X 0,Y 378.775,Z 778.548,A -85,B 0,C 180,E1 16052.828,E2 16052.828} C_VEL
LIN {X 0,Y 370.115,Z 763.557,A -85,B 0,C 180,E1 16050.253,E2 16050.253} C_VEL
LIN {X 0,Y 361.562,Z 749.799,A -85,B 0,C 180,E1 16047.415,E2 16047.415} C_VEL
LIN {X 0,Y 355.523,Z 740.554,A -85,B 0,C 180,E1 16045.174,E2 16045.174} C_VEL
LIN {X 0,Y 349.41,Z 731.532,A -85,B 0,C 180,E1 16042.636,E2 16042.636} C_VEL
LIN {X 0,Y 346.682,Z 727.716,A -85,B 0,C 180,E1 16041.397,E2 16041.397} C_VEL
LIN {X 0,Y 343.335,Z 722.863,A -85,B 0,C 180,E1 16039.743,E2 16039.743} C_VEL
LIN {X 0,Y 339.957,Z 717.938,A -85,B 0,C 180,E1 16037.899,E2 16037.899} C_VEL
LIN {X 0,Y 336.797,Z 713.583,A -85,B 0,C 180,E1 16035.982,E2 16035.982} C_VEL
LIN {X 0,Y 333.022,Z 708.416,A -85,B 0,C 180,E1 16033.322,E2 16033.322} C_VEL
LIN {X 0,Y 332.255,Z 707.102,A -85,B 0,C 180,E1 16032.69,E2 16032.69} C_VEL
LIN {X 0,Y 329.452,Z 703.853,A -85,B 0,C 180,E1 16030.226,E2 16030.226} C_VEL
LIN {X 0,Y 328.302,Z 701.694,A -85,B 0,C 180,E1 16028.935,E2 16028.935} C_VEL
LIN {X 0,Y 323.646,Z 698.414,A -85,B 0,C 180,E1 16020.354,E2 16020.354} C_VEL
LIN {X 0,Y 323.757,Z 698.546,A -85,B 0,C 180,E1 16016.459,E2 16016.459} C_VEL
LIN {X 0,Y 328.423,Z 701.803,A -85,B 0,C 180,E1 16008.408,E2 16008.408} C_VEL
LIN {X 0,Y 331.047,Z 706.054,A -85,B 0,C 180,E1 16005.75,E2 16005.75} C_VEL
LIN {X 0,Y 334.764,Z 708.692,A -85,B 0,C 180,E1 16003.025,E2 16003.025} C_VEL
LIN {X 0,Y 336.829,Z 712.204,A -85,B 0,C 180,E1 16001.57,E2 16001.57} C_VEL
LIN {X 0,Y 340.297,Z 714.98,A -85,B 0,C 180,E1 15999.595,E2 15999.595} C_VEL
LIN {X 0,Y 342.856,Z 718.857,A -85,B 0,C 180,E1 15998.172,E2 15998.172} C_VEL
LIN {X 0,Y 345.649,Z 721.378,A -85,B 0,C 180,E1 15996.833,E2 15996.833} C_VEL
LIN {X 0,Y 348.83,Z 725.625,A -85,B 0,C 180,E1 15995.351,E2 15995.351} C_VEL
LIN {X 0,Y 350.733,Z 727.555,A -85,B 0,C 180,E1 15994.548,E2 15994.548} C_VEL
LIN {X 0,Y 354.413,Z 732.05,A -85,B 0,C 180,E1 15993.049,E2 15993.049} C_VEL
LIN {X 0,Y 360.083,Z 739.337,A -85,B 0,C 180,E1 15990.926,E2 15990.926} C_VEL
LIN {X 0,Y 367.554,Z 749.078,A -85,B 0,C 180,E1 15988.422,E2 15988.422} C_VEL
LIN {X 0,Y 377.111,Z 762.445,A -85,B 0,C 180,E1 15985.565,E2 15985.565} C_VEL
LIN {X 0,Y 386.809,Z 777.188,A -85,B 0,C 180,E1 15982.966,E2 15982.966} C_VEL
LIN {X 0,Y 389.241,Z 781.367,A -85,B 0,C 180,E1 15982.345,E2 15982.345} C_VEL
LIN {X 0,Y 380.74,Z 942.738,A -85,B 0,C 180,E1 15979.131,E2 15979.131} C_VEL
LIN {X 0,Y 378.954,Z 965.608,A -85,B 0,C 180,E1 15978.409,E2 15978.409} C_VEL
LIN {X 0,Y 376.539,Z 986.118,A -85,B 0,C 180,E1 15977.52,E2 15977.52} C_VEL
LIN {X 0,Y 373.381,Z 1005.743,A -85,B 0,C 180,E1 15976.414,E2 15976.414} C_VEL
LIN {X 0,Y 369.497,Z 1025.387,A -85,B 0,C 180,E1 15975.04,E2 15975.04} C_VEL
LIN {X 0,Y 365.31,Z 1043.437,A -85,B 0,C 180,E1 15973.505,E2 15973.505} C_VEL
LIN {X 0,Y 360.411,Z 1061.473,A -85,B 0,C 180,E1 15971.637,E2 15971.637} C_VEL
LIN {X 0,Y 355.043,Z 1079.229,A -85,B 0,C 180,E1 15969.422,E2 15969.422} C_VEL
LIN {X 0,Y 349.92,Z 1094.902,A -85,B 0,C 180,E1 15967.077,E2 15967.077} C_VEL
LIN {X 0,Y 344.728,Z 1109.552,A -85,B 0,C 180,E1 15964.442,E2 15964.442} C_VEL
LIN {X 0,Y 339.827,Z 1122.822,A -85,B 0,C 180,E1 15961.581,E2 15961.581} C_VEL
LIN {X 0,Y 335.354,Z 1134.809,A -85,B 0,C 180,E1 15958.491,E2 15958.491} C_VEL
LIN {X 0,Y 331.345,Z 1145.492,A -85,B 0,C 180,E1 15955.139,E2 15955.139} C_VEL
LIN {X 0,Y 328.041,Z 1154.605,A -85,B 0,C 180,E1 15951.622,E2 15951.622} C_VEL
LIN {X 0,Y 325.437,Z 1162.39,A -85,B 0,C 180,E1 15947.892,E2 15947.892} C_VEL
LIN {X 0,Y 323.569,Z 1168.69,A -85,B 0,C 180,E1 15944,E2 15944} C_VEL
LIN {X 0,Y 322.448,Z 1173.131,A -85,B 0,C 180,E1 15940.18,E2 15940.18} C_VEL
LIN {X 0,Y 321.778,Z 1176.33,A -85,B 0,C 180,E1 15936.064,E2 15936.064} C_VEL
LIN {X 0,Y 321.546,Z 1177.887,A -85,B 0,C 180,E1 15932.317,E2 15932.317} C_VEL
LIN {X 0,Y 321.516,Z 1177.996,A -85,B 0,C 180,E1 15928.574,E2 15928.574} C_VEL
LIN {X 0,Y 321.706,Z 1176.785,A -85,B 0,C 180,E1 15924.65,E2 15924.65} C_VEL
LIN {X 0,Y 322.229,Z 1174.252,A -85,B 0,C 180,E1 15920.895,E2 15920.895} C_VEL
LIN {X 0,Y 323.168,Z 1170.153,A -85,B 0,C 180,E1 15917.056,E2 15917.056} C_VEL
LIN {X 0,Y 324.812,Z 1164.46,A -85,B 0,C 180,E1 15913.181,E2 15913.181} C_VEL
LIN {X 0,Y 327.162,Z 1157.257,A -85,B 0,C 180,E1 15909.424,E2 15909.424} C_VEL
LIN {X 0,Y 327.476,Z 1156.33,A -85,B 0,C 180,E1 15909.014,E2 15909.014} C_VEL
LIN {X 0,Y 327.532,Z 1153.689,A -85,B 0,C 180,E1 15907.74,E2 15907.74} C_VEL
LIN {X 0,Y 324.803,Z 1146.859,A -85,B 0,C 180,E1 15904.239,E2 15904.239} C_VEL
LIN {X 0,Y 325.294,Z 1144.005,A -85,B 0,C 180,E1 15903.175,E2 15903.175} C_VEL
LIN {X 0,Y 329.749,Z 1132.751,A -85,B 0,C 180,E1 15899.78,E2 15899.78} C_VEL
LIN {X 0,Y 334.725,Z 1120.231,A -85,B 0,C 180,E1 15896.66,E2 15896.66} C_VEL
LIN {X 0,Y 340.046,Z 1106.179,A -85,B 0,C 180,E1 15893.772,E2 15893.772} C_VEL
LIN {X 0,Y 345.457,Z 1091.128,A -85,B 0,C 180,E1 15891.2,E2 15891.2} C_VEL
LIN {X 0,Y 350.991,Z 1074.663,A -85,B 0,C 180,E1 15888.851,E2 15888.851} C_VEL
LIN {X 0,Y 356.066,Z 1057.936,A -85,B 0,C 180,E1 15886.863,E2 15886.863} C_VEL
LIN {X 0,Y 360.95,Z 1039.668,A -85,B 0,C 180,E1 15885.062,E2 15885.062} C_VEL
LIN {X 0,Y 365.37,Z 1020.702,A -85,B 0,C 180,E1 15883.517,E2 15883.517} C_VEL
LIN {X 0,Y 369.122,Z 1001.222,A -85,B 0,C 180,E1 15882.234,E2 15882.234} C_VEL
LIN {X 0,Y 372.251,Z 980.413,A -85,B 0,C 180,E1 15881.149,E2 15881.149} C_VEL
LIN {X 0,Y 374.647,Z 958.719,A -85,B 0,C 180,E1 15880.293,E2 15880.293} C_VEL
LIN {X 0,Y 376.072,Z 937.588,A -85,B 0,C 180,E1 15879.698,E2 15879.698} C_VEL
LIN {X 0,Y 384.316,Z 784.938,A -85,B 0,C 180,E1 15876.645,E2 15876.645} C_VEL
LIN {X 0,Y 375.468,Z 771.242,A -85,B 0,C 180,E1 15874.233,E2 15874.233} C_VEL
LIN {X 0,Y 367,Z 758.957,A -85,B 0,C 180,E1 15871.677,E2 15871.677} C_VEL
LIN {X 0,Y 359.315,Z 748.651,A -85,B 0,C 180,E1 15869.096,E2 15869.096} C_VEL
LIN {X 0,Y 355.612,Z 743.792,A -85,B 0,C 180,E1 15867.732,E2 15867.732} C_VEL
LIN {X 0,Y 351.798,Z 738.918,A -85,B 0,C 180,E1 15866.229,E2 15866.229} C_VEL
LIN {X 0,Y 347.668,Z 733.769,A -85,B 0,C 180,E1 15864.465,E2 15864.465} C_VEL
LIN {X 0,Y 344.139,Z 729.523,A -85,B 0,C 180,E1 15862.822,E2 15862.822} C_VEL
LIN {X 0,Y 343.029,Z 728.084,A -85,B 0,C 180,E1 15862.267,E2 15862.267} C_VEL
LIN {X 0,Y 339.647,Z 724.487,A -85,B 0,C 180,E1 15860.507,E2 15860.507} C_VEL
LIN {X 0,Y 338.289,Z 722.233,A -85,B 0,C 180,E1 15859.691,E2 15859.691} C_VEL
LIN {X 0,Y 335.003,Z 719.467,A -85,B 0,C 180,E1 15857.724,E2 15857.724} C_VEL
LIN {X 0,Y 332.971,Z 715.964,A -85,B 0,C 180,E1 15856.217,E2 15856.217} C_VEL
LIN {X 0,Y 329.39,Z 713.423,A -85,B 0,C 180,E1 15853.428,E2 15853.428} C_VEL
LIN {X 0,Y 327.102,Z 709.517,A -85,B 0,C 180,E1 15850.925,E2 15850.925} C_VEL
LIN {X 0,Y 322.88,Z 706.607,A -85,B 0,C 180,E1 15842.663,E2 15842.663} C_VEL
LIN {X 0,Y 323.13,Z 706.908,A -85,B 0,C 180,E1 15838.405,E2 15838.405} C_VEL
LIN {X 0,Y 327.366,Z 709.769,A -85,B 0,C 180,E1 15831.216,E2 15831.216} C_VEL
LIN {X 0,Y 329.523,Z 713.551,A -85,B 0,C 180,E1 15828.891,E2 15828.891} C_VEL
LIN {X 0,Y 331.328,Z 715.499,A -85,B 0,C 180,E1 15827.363,E2 15827.363} C_VEL
LIN {X 0,Y 334.169,Z 719.806,A -85,B 0,C 180,E1 15825.178,E2 15825.178} C_VEL
LIN {X 0,Y 335.428,Z 721.561,A -85,B 0,C 180,E1 15824.319,E2 15824.319} C_VEL
LIN {X 0,Y 339.174,Z 726.812,A -85,B 0,C 180,E1 15822.014,E2 15822.014} C_VEL
LIN {X 0,Y 343.084,Z 732.687,A -85,B 0,C 180,E1 15819.886,E2 15819.886} C_VEL
LIN {X 0,Y 347.244,Z 738.676,A -85,B 0,C 180,E1 15817.884,E2 15817.884} C_VEL
LIN {X 0,Y 355.012,Z 750.361,A -85,B 0,C 180,E1 15814.609,E2 15814.609} C_VEL
LIN {X 0,Y 363.125,Z 763.386,A -85,B 0,C 180,E1 15811.643,E2 15811.643} C_VEL
LIN {X 0,Y 371.946,Z 778.525,A -85,B 0,C 180,E1 15808.792,E2 15808.792} C_VEL
LIN {X 0,Y 380.984,Z 795.193,A -85,B 0,C 180,E1 15806.172,E2 15806.172} C_VEL
LIN {X 0,Y 383.425,Z 800.519,A -85,B 0,C 180,E1 15805.488,E2 15805.488} C_VEL
LIN {X 0,Y 384.226,Z 813.639,A -85,B 0,C 180,E1 15804.915,E2 15804.915} C_VEL
LIN {X 0,Y 372.742,Z 1028.349,A -85,B 0,C 180,E1 15800.641,E2 15800.641} C_VEL
LIN {X 0,Y 370.301,Z 1052.203,A -85,B 0,C 180,E1 15799.993,E2 15799.993} C_VEL
LIN {X 0,Y 366.826,Z 1074.059,A -85,B 0,C 180,E1 15799.204,E2 15799.204} C_VEL
LIN {X 0,Y 362.67,Z 1094.49,A -85,B 0,C 180,E1 15798.222,E2 15798.222} C_VEL
LIN {X 0,Y 357.82,Z 1115.097,A -85,B 0,C 180,E1 15796.944,E2 15796.944} C_VEL
LIN {X 0,Y 352.544,Z 1135.208,A -85,B 0,C 180,E1 15795.385,E2 15795.385} C_VEL
LIN {X 0,Y 346.954,Z 1154.51,A -85,B 0,C 180,E1 15793.53,E2 15793.53} C_VEL
LIN {X 0,Y 341.239,Z 1173.075,A -85,B 0,C 180,E1 15791.365,E2 15791.365} C_VEL
LIN {X 0,Y 335.656,Z 1190.814,A -85,B 0,C 180,E1 15788.88,E2 15788.88} C_VEL
LIN {X 0,Y 330.287,Z 1207.519,A -85,B 0,C 180,E1 15786.073,E2 15786.073} C_VEL
LIN {X 0,Y 325.533,Z 1222.723,A -85,B 0,C 180,E1 15783.018,E2 15783.018} C_VEL
LIN {X 0,Y 321.379,Z 1236.902,A -85,B 0,C 180,E1 15779.647,E2 15779.647} C_VEL
LIN {X 0,Y 317.945,Z 1250.046,A -85,B 0,C 180,E1 15775.919,E2 15775.919} C_VEL
LIN {X 0,Y 315.543,Z 1260.982,A -85,B 0,C 180,E1 15772.152,E2 15772.152} C_VEL
LIN {X 0,Y 313.989,Z 1270.479,A -85,B 0,C 180,E1 15768.183,E2 15768.183} C_VEL
LIN {X 0,Y 313.265,Z 1277.79,A -85,B 0,C 180,E1 15764.415,E2 15764.415} C_VEL
LIN {X 0,Y 313.116,Z 1283.286,A -85,B 0,C 180,E1 15760.673,E2 15760.673} C_VEL
LIN {X 0,Y 313.262,Z 1287.251,A -85,B 0,C 180,E1 15756.96,E2 15756.96} C_VEL
LIN {X 0,Y 313.471,Z 1289.336,A -85,B 0,C 180,E1 15753.657,E2 15753.657} C_VEL
LIN {X 0,Y 313.566,Z 1290.182,A -85,B 0,C 180,E1 15750.365,E2 15750.365} C_VEL
LIN {X 0,Y 313.498,Z 1289.573,A -85,B 0,C 180,E1 15746.892,E2 15746.892} C_VEL
LIN {X 0,Y 313.32,Z 1287.788,A -85,B 0,C 180,E1 15743.771,E2 15743.771} C_VEL
LIN {X 0,Y 313.129,Z 1284.234,A -85,B 0,C 180,E1 15740.071,E2 15740.071} C_VEL
LIN {X 0,Y 313.2,Z 1279.266,A -85,B 0,C 180,E1 15736.524,E2 15736.524} C_VEL
LIN {X 0,Y 313.795,Z 1272.074,A -85,B 0,C 180,E1 15732.572,E2 15732.572} C_VEL
LIN {X 0,Y 315.086,Z 1263.45,A -85,B 0,C 180,E1 15728.793,E2 15728.793} C_VEL
LIN {X 0,Y 317.241,Z 1252.887,A -85,B 0,C 180,E1 15725.019,E2 15725.019} C_VEL
LIN {X 0,Y 320.42,Z 1240.295,A -85,B 0,C 180,E1 15721.264,E2 15721.264} C_VEL
LIN {X 0,Y 324.202,Z 1227.158,A -85,B 0,C 180,E1 15717.965,E2 15717.965} C_VEL
LIN {X 0,Y 328.671,Z 1212.598,A -85,B 0,C 180,E1 15714.904,E2 15714.904} C_VEL
LIN {X 0,Y 334.164,Z 1195.3,A -85,B 0,C 180,E1 15711.84,E2 15711.84} C_VEL
LIN {X 0,Y 339.65,Z 1178.181,A -85,B 0,C 180,E1 15709.305,E2 15709.305} C_VEL
LIN {X 0,Y 345.192,Z 1160.249,A -85,B 0,C 180,E1 15707.105,E2 15707.105} C_VEL
LIN {X 0,Y 350.836,Z 1140.977,A -85,B 0,C 180,E1 15705.143,E2 15705.143} C_VEL
LIN {X 0,Y 356.266,Z 1121.148,A -85,B 0,C 180,E1 15703.493,E2 15703.493} C_VEL
LIN {X 0,Y 361.013,Z 1101.65,A -85,B 0,C 180,E1 15702.197,E2 15702.197} C_VEL
LIN {X 0,Y 365.655,Z 1079.855,A -85,B 0,C 180,E1 15701.062,E2 15701.062} C_VEL
LIN {X 0,Y 369.438,Z 1058.221,A -85,B 0,C 180,E1 15700.209,E2 15700.209} C_VEL
LIN {X 0,Y 372.102,Z 1035.736,A -85,B 0,C 180,E1 15699.542,E2 15699.542} C_VEL
LIN {X 0,Y 374.217,Z 1000.794,A -85,B 0,C 180,E1 15698.801,E2 15698.801} C_VEL
LIN {X 0,Y 384.182,Z 811.773,A -85,B 0,C 180,E1 15695.043,E2 15695.043} C_VEL
LIN {X 0,Y 383.145,Z 799.637,A -85,B 0,C 180,E1 15694.451,E2 15694.451} C_VEL
LIN {X 0,Y 374.545,Z 783.233,A -85,B 0,C 180,E1 15692.021,E2 15692.021} C_VEL
LIN {X 0,Y 366.321,Z 768.844,A -85,B 0,C 180,E1 15689.471,E2 15689.471} C_VEL
LIN {X 0,Y 357.617,Z 754.549,A -85,B 0,C 180,E1 15686.439,E2 15686.439} C_VEL
LIN {X 0,Y 351.423,Z 745.043,A -85,B 0,C 180,E1 15684.007,E2 15684.007} C_VEL
LIN {X 0,Y 345.365,Z 735.873,A -85,B 0,C 180,E1 15681.305,E2 15681.305} C_VEL
LIN {X 0,Y 340.96,Z 729.644,A -85,B 0,C 180,E1 15679.085,E2 15679.085} C_VEL
LIN {X 0,Y 338.118,Z 725.332,A -85,B 0,C 180,E1 15677.466,E2 15677.466} C_VEL
LIN {X 0,Y 334.932,Z 720.714,A -85,B 0,C 180,E1 15675.452,E2 15675.452} C_VEL
LIN {X 0,Y 331.647,Z 716.266,A -85,B 0,C 180,E1 15673.068,E2 15673.068} C_VEL
LIN {X 0,Y 330.641,Z 714.625,A -85,B 0,C 180,E1 15672.22,E2 15672.22} C_VEL
LIN {X 0,Y 327.974,Z 711.234,A -85,B 0,C 180,E1 15669.741,E2 15669.741} C_VEL
LIN {X 0,Y 327.17,Z 709.574,A -85,B 0,C 180,E1 15668.789,E2 15668.789} C_VEL
LIN {X 0,Y 322.671,Z 706.357,A -85,B 0,C 180,E1 15660.355,E2 15660.355} C_VEL
LIN {X 0,Y 322.783,Z 706.497,A -85,B 0,C 180,E1 15656.448,E2 15656.448} C_VEL
LIN {X 0,Y 327.373,Z 709.785,A -85,B 0,C 180,E1 15648.46,E2 15648.46} C_VEL
LIN {X 0,Y 329.492,Z 713.544,A -85,B 0,C 180,E1 15646.219,E2 15646.219} C_VEL
LIN {X 0,Y 333.194,Z 716.352,A -85,B 0,C 180,E1 15643.391,E2 15643.391} C_VEL
LIN {X 0,Y 335.475,Z 720.049,A -85,B 0,C 180,E1 15641.763,E2 15641.763} C_VEL
LIN {X 0,Y 338.62,Z 722.736,A -85,B 0,C 180,E1 15639.924,E2 15639.924} C_VEL
LIN {X 0,Y 341.433,Z 726.728,A -85,B 0,C 180,E1 15638.347,E2 15638.347} C_VEL
LIN {X 0,Y 343.775,Z 728.955,A -85,B 0,C 180,E1 15637.197,E2 15637.197} C_VEL
LIN {X 0,Y 347.178,Z 733.345,A -85,B 0,C 180,E1 15635.589,E2 15635.589} C_VEL
LIN {X 0,Y 348.858,Z 735.27,A -85,B 0,C 180,E1 15634.856,E2 15634.856} C_VEL
LIN {X 0,Y 353.472,Z 741.051,A -85,B 0,C 180,E1 15632.953,E2 15632.953} C_VEL
LIN {X 0,Y 357.989,Z 746.948,A -85,B 0,C 180,E1 15631.243,E2 15631.243} C_VEL
LIN {X 0,Y 364.825,Z 755.982,A -85,B 0,C 180,E1 15628.894,E2 15628.894} C_VEL
LIN {X 0,Y 374.1,Z 769.203,A -85,B 0,C 180,E1 15626.041,E2 15626.041} C_VEL
LIN {X 0,Y 383.419,Z 783.595,A -85,B 0,C 180,E1 15623.472,E2 15623.472} C_VEL
LIN {X 0,Y 384.312,Z 785.319,A -85,B 0,C 180,E1 15623.229,E2 15623.229} C_VEL
LIN {X 0,Y 375.641,Z 943.713,A -85,B 0,C 180,E1 15620.054,E2 15620.054} C_VEL
LIN {X 0,Y 373.792,Z 966.758,A -85,B 0,C 180,E1 15619.323,E2 15619.323} C_VEL
LIN {X 0,Y 371.264,Z 987.518,A -85,B 0,C 180,E1 15618.417,E2 15618.417} C_VEL
LIN {X 0,Y 367.995,Z 1007.141,A -85,B 0,C 180,E1 15617.302,E2 15617.302} C_VEL
LIN {X 0,Y 363.972,Z 1026.785,A -85,B 0,C 180,E1 15615.917,E2 15615.917} C_VEL
LIN {X 0,Y 359.64,Z 1044.801,A -85,B 0,C 180,E1 15614.373,E2 15614.373} C_VEL
LIN {X 0,Y 354.551,Z 1062.87,A -85,B 0,C 180,E1 15612.484,E2 15612.484} C_VEL
LIN {X 0,Y 348.971,Z 1080.628,A -85,B 0,C 180,E1 15610.246,E2 15610.246} C_VEL
LIN {X 0,Y 343.453,Z 1096.782,A -85,B 0,C 180,E1 15607.791,E2 15607.791} C_VEL
LIN {X 0,Y 338.214,Z 1110.955,A -85,B 0,C 180,E1 15605.202,E2 15605.202} C_VEL
LIN {X 0,Y 333.082,Z 1124.227,A -85,B 0,C 180,E1 15602.297,E2 15602.297} C_VEL
LIN {X 0,Y 328.383,Z 1136.215,A -85,B 0,C 180,E1 15599.154,E2 15599.154} C_VEL
LIN {X 0,Y 324.176,Z 1146.833,A -85,B 0,C 180,E1 15595.76,E2 15595.76} C_VEL
LIN {X 0,Y 320.665,Z 1155.97,A -85,B 0,C 180,E1 15592.165,E2 15592.165} C_VEL
LIN {X 0,Y 317.871,Z 1163.795,A -85,B 0,C 180,E1 15588.333,E2 15588.333} C_VEL
LIN {X 0,Y 315.896,Z 1170.002,A -85,B 0,C 180,E1 15584.41,E2 15584.41} C_VEL
LIN {X 0,Y 314.654,Z 1174.529,A -85,B 0,C 180,E1 15580.435,E2 15580.435} C_VEL
LIN {X 0,Y 313.928,Z 1177.724,A -85,B 0,C 180,E1 15576.217,E2 15576.217} C_VEL
LIN {X 0,Y 313.671,Z 1179.278,A -85,B 0,C 180,E1 15572.375,E2 15572.375} C_VEL
LIN {X 0,Y 313.638,Z 1179.386,A -85,B 0,C 180,E1 15568.539,E2 15568.539} C_VEL
LIN {X 0,Y 313.848,Z 1178.177,A -85,B 0,C 180,E1 15564.516,E2 15564.516} C_VEL
LIN {X 0,Y 314.415,Z 1175.649,A -85,B 0,C 180,E1 15560.667,E2 15560.667} C_VEL
LIN {X 0,Y 315.452,Z 1171.481,A -85,B 0,C 180,E1 15556.674,E2 15556.674} C_VEL
LIN {X 0,Y 317.299,Z 1165.547,A -85,B 0,C 180,E1 15552.581,E2 15552.581} C_VEL
LIN {X 0,Y 319.902,Z 1158.175,A -85,B 0,C 180,E1 15548.696,E2 15548.696} C_VEL
LIN {X 0,Y 323.338,Z 1149.037,A -85,B 0,C 180,E1 15544.936,E2 15544.936} C_VEL
LIN {X 0,Y 325.294,Z 1144.005,A -85,B 0,C 180,E1 15543.175,E2 15543.175} C_VEL
LIN {X 0,Y 325.859,Z 1140.686,A -85,B 0,C 180,E1 15541.943,E2 15541.943} C_VEL
LIN {X 0,Y 324.473,Z 1132.465,A -85,B 0,C 180,E1 15538.713,E2 15538.713} C_VEL
LIN {X 0,Y 325.288,Z 1128.46,A -85,B 0,C 180,E1 15537.55,E2 15537.55} C_VEL
LIN {X 0,Y 330.648,Z 1115.304,A -85,B 0,C 180,E1 15534.509,E2 15534.509} C_VEL
LIN {X 0,Y 336.173,Z 1101.051,A -85,B 0,C 180,E1 15531.784,E2 15531.784} C_VEL
LIN {X 0,Y 342.034,Z 1084.937,A -85,B 0,C 180,E1 15529.212,E2 15529.212} C_VEL
LIN {X 0,Y 347.574,Z 1068.411,A -85,B 0,C 180,E1 15527.019,E2 15527.019} C_VEL
LIN {X 0,Y 352.739,Z 1050.962,A -85,B 0,C 180,E1 15525.107,E2 15525.107} C_VEL
LIN {X 0,Y 357.7,Z 1032.011,A -85,B 0,C 180,E1 15523.386,E2 15523.386} C_VEL
LIN {X 0,Y 362.021,Z 1012.605,A -85,B 0,C 180,E1 15521.942,E2 15521.942} C_VEL
LIN {X 0,Y 365.581,Z 992.411,A -85,B 0,C 180,E1 15520.75,E2 15520.75} C_VEL
LIN {X 0,Y 368.505,Z 970.67,A -85,B 0,C 180,E1 15519.749,E2 15519.749} C_VEL
LIN {X 0,Y 370.449,Z 949.708,A -85,B 0,C 180,E1 15519.032,E2 15519.032} C_VEL
LIN {X 0,Y 372.627,Z 909.433,A -85,B 0,C 180,E1 15518.145,E2 15518.145} C_VEL
LIN {X 0,Y 379.528,Z 789.064,A -85,B 0,C 180,E1 15515.751,E2 15515.751} C_VEL
LIN {X 0,Y 370.522,Z 774.97,A -85,B 0,C 180,E1 15513.17,E2 15513.17} C_VEL
LIN {X 0,Y 361.48,Z 761.879,A -85,B 0,C 180,E1 15510.272,E2 15510.272} C_VEL
LIN {X 0,Y 353.362,Z 751.034,A -85,B 0,C 180,E1 15507.32,E2 15507.32} C_VEL
LIN {X 0,Y 349.539,Z 746.095,A -85,B 0,C 180,E1 15505.773,E2 15505.773} C_VEL
LIN {X 0,Y 345.49,Z 741,A -85,B 0,C 180,E1 15503.992,E2 15503.992} C_VEL
LIN {X 0,Y 341.903,Z 736.419,A -85,B 0,C 180,E1 15502.254,E2 15502.254} C_VEL
LIN {X 0,Y 337.613,Z 731.532,A -85,B 0,C 180,E1 15499.958,E2 15499.958} C_VEL
LIN {X 0,Y 336.475,Z 729.785,A -85,B 0,C 180,E1 15499.26,E2 15499.26} C_VEL
LIN {X 0,Y 333.178,Z 726.692,A -85,B 0,C 180,E1 15497.194,E2 15497.194} C_VEL
LIN {X 0,Y 331.541,Z 723.735,A -85,B 0,C 180,E1 15495.929,E2 15495.929} C_VEL
LIN {X 0,Y 328.053,Z 721.121,A -85,B 0,C 180,E1 15493.125,E2 15493.125} C_VEL
LIN {X 0,Y 325.985,Z 717.398,A -85,B 0,C 180,E1 15490.784,E2 15490.784} C_VEL
LIN {X 0,Y 321.885,Z 714.525,A -85,B 0,C 180,E1 15482.493,E2 15482.493} C_VEL
LIN {X 0,Y 322.199,Z 714.909,A -85,B 0,C 180,E1 15478.222,E2 15478.222} C_VEL
LIN {X 0,Y 326.157,Z 717.607,A -85,B 0,C 180,E1 15471.45,E2 15471.45} C_VEL
LIN {X 0,Y 328.266,Z 721.348,A -85,B 0,C 180,E1 15469.115,E2 15469.115} C_VEL
LIN {X 0,Y 329.878,Z 723.155,A -85,B 0,C 180,E1 15467.706,E2 15467.706} C_VEL
LIN {X 0,Y 332.708,Z 727.489,A -85,B 0,C 180,E1 15465.467,E2 15465.467} C_VEL
LIN {X 0,Y 334.493,Z 730.281,A -85,B 0,C 180,E1 15464.216,E2 15464.216} C_VEL
LIN {X 0,Y 337.335,Z 734.191,A -85,B 0,C 180,E1 15462.447,E2 15462.447} C_VEL
LIN {X 0,Y 341.226,Z 740.19,A -85,B 0,C 180,E1 15460.263,E2 15460.263} C_VEL
LIN {X 0,Y 345.474,Z 746.435,A -85,B 0,C 180,E1 15458.168,E2 15458.168} C_VEL
LIN {X 0,Y 352.746,Z 757.747,A -85,B 0,C 180,E1 15455.018,E2 15455.018} C_VEL
LIN {X 0,Y 360.213,Z 769.943,A -85,B 0,C 180,E1 15452.204,E2 15452.204} C_VEL
LIN {X 0,Y 368.69,Z 784.816,A -85,B 0,C 180,E1 15449.37,E2 15449.37} C_VEL
LIN {X 0,Y 377.498,Z 801.398,A -85,B 0,C 180,E1 15446.729,E2 15446.729} C_VEL
LIN {X 0,Y 378.913,Z 804.774,A -85,B 0,C 180,E1 15446.309,E2 15446.309} C_VEL
LIN {X 0,Y 379.455,Z 814.976,A -85,B 0,C 180,E1 15445.864,E2 15445.864} C_VEL
LIN {X 0,Y 367.599,Z 1027.696,A -85,B 0,C 180,E1 15441.601,E2 15441.601} C_VEL
LIN {X 0,Y 365.111,Z 1050.995,A -85,B 0,C 180,E1 15440.961,E2 15440.961} C_VEL
LIN {X 0,Y 361.574,Z 1072.634,A -85,B 0,C 180,E1 15440.178,E2 15440.178} C_VEL
LIN {X 0,Y 357.277,Z 1093.055,A -85,B 0,C 180,E1 15439.199,E2 15439.199} C_VEL
LIN {X 0,Y 352.285,Z 1113.548,A -85,B 0,C 180,E1 15437.929,E2 15437.929} C_VEL
LIN {X 0,Y 346.787,Z 1133.754,A -85,B 0,C 180,E1 15436.358,E2 15436.358} C_VEL
LIN {X 0,Y 341.21,Z 1152.283,A -85,B 0,C 180,E1 15434.571,E2 15434.571} C_VEL
LIN {X 0,Y 334.98,Z 1171.665,A -85,B 0,C 180,E1 15432.304,E2 15432.304} C_VEL
LIN {X 0,Y 329.252,Z 1189.037,A -85,B 0,C 180,E1 15429.847,E2 15429.847} C_VEL
LIN {X 0,Y 323.667,Z 1205.552,A -85,B 0,C 180,E1 15427.04,E2 15427.04} C_VEL
LIN {X 0,Y 318.638,Z 1220.747,A -85,B 0,C 180,E1 15423.954,E2 15423.954} C_VEL
LIN {X 0,Y 314.28,Z 1234.718,A -85,B 0,C 180,E1 15420.598,E2 15420.598} C_VEL
LIN {X 0,Y 310.554,Z 1247.943,A -85,B 0,C 180,E1 15416.791,E2 15416.791} C_VEL
LIN {X 0,Y 307.918,Z 1258.995,A -85,B 0,C 180,E1 15412.933,E2 15412.933} C_VEL
LIN {X 0,Y 306.152,Z 1268.91,A -85,B 0,C 180,E1 15408.72,E2 15408.72} C_VEL
LIN {X 0,Y 305.352,Z 1276.348,A -85,B 0,C 180,E1 15404.797,E2 15404.797} C_VEL
LIN {X 0,Y 305.184,Z 1281.861,A -85,B 0,C 180,E1 15400.954,E2 15400.954} C_VEL
LIN {X 0,Y 305.343,Z 1285.839,A -85,B 0,C 180,E1 15397.148,E2 15397.148} C_VEL
LIN {X 0,Y 305.578,Z 1287.94,A -85,B 0,C 180,E1 15393.752,E2 15393.752} C_VEL
LIN {X 0,Y 305.687,Z 1288.791,A -85,B 0,C 180,E1 15390.375,E2 15390.375} C_VEL
LIN {X 0,Y 305.608,Z 1288.179,A -85,B 0,C 180,E1 15386.812,E2 15386.812} C_VEL
LIN {X 0,Y 305.411,Z 1286.383,A -85,B 0,C 180,E1 15383.609,E2 15383.609} C_VEL
LIN {X 0,Y 305.194,Z 1282.811,A -85,B 0,C 180,E1 15379.81,E2 15379.81} C_VEL
LIN {X 0,Y 305.272,Z 1277.826,A -85,B 0,C 180,E1 15376.167,E2 15376.167} C_VEL
LIN {X 0,Y 305.92,Z 1270.615,A -85,B 0,C 180,E1 15372.108,E2 15372.108} C_VEL
LIN {X 0,Y 307.326,Z 1261.977,A -85,B 0,C 180,E1 15368.23,E2 15368.23} C_VEL
LIN {X 0,Y 309.651,Z 1251.404,A -85,B 0,C 180,E1 15364.363,E2 15364.363} C_VEL
LIN {X 0,Y 313.037,Z 1238.859,A -85,B 0,C 180,E1 15360.536,E2 15360.536} C_VEL
LIN {X 0,Y 317.066,Z 1225.664,A -85,B 0,C 180,E1 15357.154,E2 15357.154} C_VEL
LIN {X 0,Y 321.791,Z 1211.104,A -85,B 0,C 180,E1 15354.039,E2 15354.039} C_VEL
LIN {X 0,Y 327.412,Z 1194.35,A -85,B 0,C 180,E1 15351.019,E2 15351.019} C_VEL
LIN {X 0,Y 333.134,Z 1177.335,A -85,B 0,C 180,E1 15348.449,E2 15348.449} C_VEL
LIN {X 0,Y 339.127,Z 1158.773,A -85,B 0,C 180,E1 15346.145,E2 15346.145} C_VEL
LIN {X 0,Y 345.141,Z 1139.093,A -85,B 0,C 180,E1 15344.135,E2 15344.135} C_VEL
LIN {X 0,Y 350.687,Z 1119.57,A -85,B 0,C 180,E1 15342.51,E2 15342.51} C_VEL
LIN {X 0,Y 355.658,Z 1099.861,A -85,B 0,C 180,E1 15341.2,E2 15341.2} C_VEL
LIN {X 0,Y 360.366,Z 1078.411,A -85,B 0,C 180,E1 15340.088,E2 15340.088} C_VEL
LIN {X 0,Y 364.272,Z 1056.642,A -85,B 0,C 180,E1 15339.23,E2 15339.23} C_VEL
LIN {X 0,Y 366.991,Z 1034.289,A -85,B 0,C 180,E1 15338.565,E2 15338.565} C_VEL
LIN {X 0,Y 369.186,Z 999.338,A -85,B 0,C 180,E1 15337.819,E2 15337.819} C_VEL
LIN {X 0,Y 379.405,Z 813.167,A -85,B 0,C 180,E1 15334.094,E2 15334.094} C_VEL
LIN {X 0,Y 378.648,Z 803.913,A -85,B 0,C 180,E1 15333.632,E2 15333.632} C_VEL
LIN {X 0,Y 370.335,Z 787.816,A -85,B 0,C 180,E1 15331.178,E2 15331.178} C_VEL
LIN {X 0,Y 361.66,Z 772.453,A -85,B 0,C 180,E1 15328.348,E2 15328.348} C_VEL
LIN {X 0,Y 354.33,Z 760.418,A -85,B 0,C 180,E1 15325.667,E2 15325.667} C_VEL
LIN {X 0,Y 348.959,Z 751.925,A -85,B 0,C 180,E1 15323.47,E2 15323.47} C_VEL
LIN {X 0,Y 343.215,Z 743.031,A -85,B 0,C 180,E1 15320.818,E2 15320.818} C_VEL
LIN {X 0,Y 338.78,Z 736.594,A -85,B 0,C 180,E1 15318.498,E2 15318.498} C_VEL
LIN {X 0,Y 336.299,Z 732.721,A -85,B 0,C 180,E1 15317.028,E2 15317.028} C_VEL
LIN {X 0,Y 332.535,Z 727.352,A -85,B 0,C 180,E1 15314.54,E2 15314.54} C_VEL
LIN {X 0,Y 329.658,Z 722.817,A -85,B 0,C 180,E1 15312.257,E2 15312.257} C_VEL
LIN {X 0,Y 326.593,Z 718.77,A -85,B 0,C 180,E1 15309.338,E2 15309.338} C_VEL
LIN {X 0,Y 325.886,Z 717.326,A -85,B 0,C 180,E1 15308.468,E2 15308.468} C_VEL
LIN {X 0,Y 321.652,Z 714.245,A -85,B 0,C 180,E1 15300,E2 15300} C_VEL
LIN {X 0,Y 321.881,Z 714.558,A -85,B 0,C 180,E1 15296.081,E2 15296.081} C_VEL
LIN {X 0,Y 326.167,Z 717.607,A -85,B 0,C 180,E1 15288.685,E2 15288.685} C_VEL
LIN {X 0,Y 328.053,Z 721.133,A -85,B 0,C 180,E1 15286.606,E2 15286.606} C_VEL
LIN {X 0,Y 331.692,Z 724.1,A -85,B 0,C 180,E1 15283.719,E2 15283.719} C_VEL
LIN {X 0,Y 334.254,Z 728.022,A -85,B 0,C 180,E1 15281.874,E2 15281.874} C_VEL
LIN {X 0,Y 336.937,Z 730.394,A -85,B 0,C 180,E1 15280.272,E2 15280.272} C_VEL
LIN {X 0,Y 340.016,Z 734.585,A -85,B 0,C 180,E1 15278.524,E2 15278.524} C_VEL
LIN {X 0,Y 341.917,Z 736.506,A -85,B 0,C 180,E1 15277.566,E2 15277.566} C_VEL
LIN {X 0,Y 345.532,Z 741.06,A -85,B 0,C 180,E1 15275.829,E2 15275.829} C_VEL
LIN {X 0,Y 351.269,Z 748.349,A -85,B 0,C 180,E1 15273.364,E2 15273.364} C_VEL
LIN {X 0,Y 355.909,Z 754.527,A -85,B 0,C 180,E1 15271.564,E2 15271.564} C_VEL
LIN {X 0,Y 362.439,Z 763.365,A -85,B 0,C 180,E1 15269.266,E2 15269.266} C_VEL
LIN {X 0,Y 371.128,Z 775.976,A -85,B 0,C 180,E1 15266.522,E2 15266.522} C_VEL
LIN {X 0,Y 379.482,Z 789.078,A -85,B 0,C 180,E1 15264.142,E2 15264.142} C_VEL
LIN {X 0,Y 370.636,Z 944.774,A -85,B 0,C 180,E1 15261,E2 15261} C_VEL
LIN {X 0,Y 368.784,Z 967.4,A -85,B 0,C 180,E1 15260.282,E2 15260.282} C_VEL
LIN {X 0,Y 366.198,Z 988.174,A -85,B 0,C 180,E1 15259.378,E2 15259.378} C_VEL
LIN {X 0,Y 362.7,Z 1008.54,A -85,B 0,C 180,E1 15258.216,E2 15258.216} C_VEL
LIN {X 0,Y 358.535,Z 1028.182,A -85,B 0,C 180,E1 15256.822,E2 15256.822} C_VEL
LIN {X 0,Y 353.803,Z 1047.099,A -85,B 0,C 180,E1 15255.179,E2 15255.179} C_VEL
LIN {X 0,Y 348.56,Z 1064.971,A -85,B 0,C 180,E1 15253.28,E2 15253.28} C_VEL
LIN {X 0,Y 342.974,Z 1082.027,A -85,B 0,C 180,E1 15251.1,E2 15251.1} C_VEL
LIN {X 0,Y 337.414,Z 1097.705,A -85,B 0,C 180,E1 15248.7,E2 15248.7} C_VEL
LIN {X 0,Y 331.763,Z 1112.359,A -85,B 0,C 180,E1 15245.992,E2 15245.992} C_VEL
LIN {X 0,Y 326.392,Z 1125.632,A -85,B 0,C 180,E1 15243.043,E2 15243.043} C_VEL
LIN {X 0,Y 321.456,Z 1137.621,A -85,B 0,C 180,E1 15239.845,E2 15239.845} C_VEL
LIN {X 0,Y 317.038,Z 1148.195,A -85,B 0,C 180,E1 15236.402,E2 15236.402} C_VEL
LIN {X 0,Y 313.302,Z 1157.377,A -85,B 0,C 180,E1 15232.715,E2 15232.715} C_VEL
LIN {X 0,Y 310.324,Z 1165.202,A -85,B 0,C 180,E1 15228.795,E2 15228.795} C_VEL
LIN {X 0,Y 308.238,Z 1171.317,A -85,B 0,C 180,E1 15224.838,E2 15224.838} C_VEL
LIN {X 0,Y 306.908,Z 1175.748,A -85,B 0,C 180,E1 15220.891,E2 15220.891} C_VEL
LIN {X 0,Y 306.132,Z 1178.921,A -85,B 0,C 180,E1 15216.752,E2 15216.752} C_VEL
LIN {X 0,Y 305.813,Z 1180.491,A -85,B 0,C 180,E1 15212.999,E2 15212.999} C_VEL
LIN {X 0,Y 305.76,Z 1180.815,A -85,B 0,C 180,E1 15208.876,E2 15208.876} C_VEL
LIN {X 0,Y 305.953,Z 1179.868,A -85,B 0,C 180,E1 15204.938,E2 15204.938} C_VEL
LIN {X 0,Y 306.487,Z 1177.459,A -85,B 0,C 180,E1 15200.991,E2 15200.991} C_VEL
LIN {X 0,Y 307.617,Z 1173.267,A -85,B 0,C 180,E1 15196.658,E2 15196.658} C_VEL
LIN {X 0,Y 309.409,Z 1167.899,A -85,B 0,C 180,E1 15192.705,E2 15192.705} C_VEL
LIN {X 0,Y 311.99,Z 1160.796,A -85,B 0,C 180,E1 15188.769,E2 15188.769} C_VEL
LIN {X 0,Y 315.351,Z 1152.32,A -85,B 0,C 180,E1 15185.059,E2 15185.059} C_VEL
LIN {X 0,Y 319.639,Z 1142.024,A -85,B 0,C 180,E1 15181.407,E2 15181.407} C_VEL
LIN {X 0,Y 324.279,Z 1130.902,A -85,B 0,C 180,E1 15178.181,E2 15178.181} C_VEL
LIN {X 0,Y 325.288,Z 1128.46,A -85,B 0,C 180,E1 15177.55,E2 15177.55} C_VEL
LIN {X 0,Y 326.187,Z 1124.389,A -85,B 0,C 180,E1 15176.406,E2 15176.406} C_VEL
LIN {X 0,Y 325.884,Z 1114.391,A -85,B 0,C 180,E1 15173.341,E2 15173.341} C_VEL
LIN {X 0,Y 327.093,Z 1109.666,A -85,B 0,C 180,E1 15172.268,E2 15172.268} C_VEL
LIN {X 0,Y 333.069,Z 1094.441,A -85,B 0,C 180,E1 15169.579,E2 15169.579} C_VEL
LIN {X 0,Y 338.829,Z 1078.717,A -85,B 0,C 180,E1 15167.259,E2 15167.259} C_VEL
LIN {X 0,Y 344.488,Z 1061.415,A -85,B 0,C 180,E1 15165.149,E2 15165.149} C_VEL
LIN {X 0,Y 349.685,Z 1043.483,A -85,B 0,C 180,E1 15163.333,E2 15163.333} C_VEL
LIN {X 0,Y 354.544,Z 1024.213,A -85,B 0,C 180,E1 15161.725,E2 15161.725} C_VEL
LIN {X 0,Y 358.547,Z 1004.857,A -85,B 0,C 180,E1 15160.423,E2 15160.423} C_VEL
LIN {X 0,Y 361.99,Z 983.729,A -85,B 0,C 180,E1 15159.296,E2 15159.296} C_VEL
LIN {X 0,Y 364.561,Z 962.269,A -85,B 0,C 180,E1 15158.425,E2 15158.425} C_VEL
LIN {X 0,Y 366.122,Z 940.969,A -85,B 0,C 180,E1 15157.808,E2 15157.808} C_VEL
LIN {X 0,Y 374.772,Z 793.051,A -85,B 0,C 180,E1 15154.816,E2 15154.816} C_VEL
LIN {X 0,Y 365.907,Z 779.236,A -85,B 0,C 180,E1 15152.152,E2 15152.152} C_VEL
LIN {X 0,Y 358.397,Z 768.255,A -85,B 0,C 180,E1 15149.637,E2 15149.637} C_VEL
LIN {X 0,Y 350.975,Z 758.094,A -85,B 0,C 180,E1 15146.843,E2 15146.843} C_VEL
LIN {X 0,Y 347.031,Z 752.964,A -85,B 0,C 180,E1 15145.195,E2 15145.195} C_VEL
LIN {X 0,Y 343.338,Z 748.213,A -85,B 0,C 180,E1 15143.514,E2 15143.514} C_VEL
LIN {X 0,Y 339.219,Z 742.964,A -85,B 0,C 180,E1 15141.438,E2 15141.438} C_VEL
LIN {X 0,Y 335.742,Z 738.796,A -85,B 0,C 180,E1 15139.484,E2 15139.484} C_VEL
LIN {X 0,Y 334.683,Z 737.313,A -85,B 0,C 180,E1 15138.823,E2 15138.823} C_VEL
LIN {X 0,Y 331.497,Z 734.072,A -85,B 0,C 180,E1 15136.741,E2 15136.741} C_VEL
LIN {X 0,Y 329.834,Z 731.352,A -85,B 0,C 180,E1 15135.431,E2 15135.431} C_VEL
LIN {X 0,Y 326.467,Z 728.477,A -85,B 0,C 180,E1 15132.56,E2 15132.56} C_VEL
LIN {X 0,Y 324.721,Z 725.159,A -85,B 0,C 180,E1 15130.467,E2 15130.467} C_VEL
LIN {X 0,Y 320.892,Z 722.446,A -85,B 0,C 180,E1 15122.322,E2 15122.322} C_VEL
LIN {X 0,Y 321.271,Z 722.912,A -85,B 0,C 180,E1 15118.038,E2 15118.038} C_VEL
LIN {X 0,Y 324.948,Z 725.485,A -85,B 0,C 180,E1 15111.685,E2 15111.685} C_VEL
LIN {X 0,Y 327.105,Z 729.248,A -85,B 0,C 180,E1 15109.254,E2 15109.254} C_VEL
LIN {X 0,Y 328.44,Z 730.81,A -85,B 0,C 180,E1 15108.053,E2 15108.053} C_VEL
LIN {X 0,Y 331.375,Z 735.301,A -85,B 0,C 180,E1 15105.676,E2 15105.676} C_VEL
LIN {X 0,Y 335.646,Z 741.803,A -85,B 0,C 180,E1 15102.803,E2 15102.803} C_VEL
LIN {X 0,Y 339.31,Z 747.564,A -85,B 0,C 180,E1 15100.685,E2 15100.685} C_VEL
LIN {X 0,Y 344.135,Z 754.756,A -85,B 0,C 180,E1 15098.257,E2 15098.257} C_VEL
LIN {X 0,Y 350.866,Z 765.741,A -85,B 0,C 180,E1 15095.28,E2 15095.28} C_VEL
LIN {X 0,Y 357.535,Z 776.859,A -85,B 0,C 180,E1 15092.702,E2 15092.702} C_VEL
LIN {X 0,Y 365.525,Z 791.208,A -85,B 0,C 180,E1 15089.939,E2 15089.939} C_VEL
LIN {X 0,Y 373.989,Z 807.492,A -85,B 0,C 180,E1 15087.314,E2 15087.314} C_VEL
LIN {X 0,Y 374.488,Z 809.257,A -85,B 0,C 180,E1 15087.141,E2 15087.141} C_VEL
LIN {X 0,Y 374.777,Z 816.535,A -85,B 0,C 180,E1 15086.833,E2 15086.833} C_VEL
LIN {X 0,Y 362.567,Z 1026.974,A -85,B 0,C 180,E1 15082.59,E2 15082.59} C_VEL
LIN {X 0,Y 360.013,Z 1049.893,A -85,B 0,C 180,E1 15081.953,E2 15081.953} C_VEL
LIN {X 0,Y 356.277,Z 1071.962,A -85,B 0,C 180,E1 15081.146,E2 15081.146} C_VEL
LIN {X 0,Y 351.705,Z 1092.932,A -85,B 0,C 180,E1 15080.135,E2 15080.135} C_VEL
LIN {X 0,Y 346.527,Z 1113.238,A -85,B 0,C 180,E1 15078.856,E2 15078.856} C_VEL
LIN {X 0,Y 340.872,Z 1133.138,A -85,B 0,C 180,E1 15077.286,E2 15077.286} C_VEL
LIN {X 0,Y 335.043,Z 1151.764,A -85,B 0,C 180,E1 15075.469,E2 15075.469} C_VEL
LIN {X 0,Y 328.624,Z 1170.831,A -85,B 0,C 180,E1 15073.201,E2 15073.201} C_VEL
LIN {X 0,Y 322.451,Z 1188.63,A -85,B 0,C 180,E1 15070.628,E2 15070.628} C_VEL
LIN {X 0,Y 316.475,Z 1205.548,A -85,B 0,C 180,E1 15067.685,E2 15067.685} C_VEL
LIN {X 0,Y 311.099,Z 1220.921,A -85,B 0,C 180,E1 15064.447,E2 15064.447} C_VEL
LIN {X 0,Y 306.364,Z 1235.314,A -85,B 0,C 180,E1 15060.822,E2 15060.822} C_VEL
LIN {X 0,Y 302.727,Z 1247.654,A -85,B 0,C 180,E1 15057.115,E2 15057.115} C_VEL
LIN {X 0,Y 299.957,Z 1258.76,A -85,B 0,C 180,E1 15053.075,E2 15053.075} C_VEL
LIN {X 0,Y 298.235,Z 1267.961,A -85,B 0,C 180,E1 15048.977,E2 15048.977} C_VEL
LIN {X 0,Y 297.422,Z 1275.205,A -85,B 0,C 180,E1 15045.002,E2 15045.002} C_VEL
LIN {X 0,Y 297.254,Z 1280.435,A -85,B 0,C 180,E1 15041.25,E2 15041.25} C_VEL
LIN {X 0,Y 297.421,Z 1284.43,A -85,B 0,C 180,E1 15037.339,E2 15037.339} C_VEL
LIN {X 0,Y 297.685,Z 1286.544,A -85,B 0,C 180,E1 15033.852,E2 15033.852} C_VEL
LIN {X 0,Y 297.806,Z 1287.376,A -85,B 0,C 180,E1 15030.577,E2 15030.577} C_VEL
LIN {X 0,Y 297.728,Z 1286.864,A -85,B 0,C 180,E1 15026.92,E2 15026.92} C_VEL
LIN {X 0,Y 297.511,Z 1285.114,A -85,B 0,C 180,E1 15023.633,E2 15023.633} C_VEL
LIN {X 0,Y 297.261,Z 1281.626,A -85,B 0,C 180,E1 15019.731,E2 15019.731} C_VEL
LIN {X 0,Y 297.328,Z 1276.679,A -85,B 0,C 180,E1 15015.989,E2 15015.989} C_VEL
LIN {X 0,Y 297.956,Z 1269.957,A -85,B 0,C 180,E1 15012.018,E2 15012.018} C_VEL
LIN {X 0,Y 299.396,Z 1261.42,A -85,B 0,C 180,E1 15008.036,E2 15008.036} C_VEL
LIN {X 0,Y 301.794,Z 1251.062,A -85,B 0,C 180,E1 15004.068,E2 15004.068} C_VEL
LIN {X 0,Y 305.194,Z 1239.115,A -85,B 0,C 180,E1 15000.247,E2 15000.247} C_VEL
LIN {X 0,Y 309.471,Z 1225.693,A -85,B 0,C 180,E1 14996.686,E2 14996.686} C_VEL
LIN {X 0,Y 314.67,Z 1210.517,A -85,B 0,C 180,E1 14993.32,E2 14993.32} C_VEL
LIN {X 0,Y 320.545,Z 1193.938,A -85,B 0,C 180,E1 14990.251,E2 14990.251} C_VEL
LIN {X 0,Y 326.485,Z 1177.045,A -85,B 0,C 180,E1 14987.645,E2 14987.645} C_VEL
LIN {X 0,Y 332.7,Z 1158.693,A -85,B 0,C 180,E1 14985.314,E2 14985.314} C_VEL
LIN {X 0,Y 339.049,Z 1138.887,A -85,B 0,C 180,E1 14983.249,E2 14983.249} C_VEL
LIN {X 0,Y 344.88,Z 1119.26,A -85,B 0,C 180,E1 14981.586,E2 14981.586} C_VEL
LIN {X 0,Y 350.24,Z 1098.752,A -85,B 0,C 180,E1 14980.215,E2 14980.215} C_VEL
LIN {X 0,Y 355.101,Z 1077.381,A -85,B 0,C 180,E1 14979.103,E2 14979.103} C_VEL
LIN {X 0,Y 359.142,Z 1055.595,A -85,B 0,C 180,E1 14978.241,E2 14978.241} C_VEL
LIN {X 0,Y 361.953,Z 1033.172,A -85,B 0,C 180,E1 14977.57,E2 14977.57} C_VEL
LIN {X 0,Y 364.173,Z 999.557,A -85,B 0,C 180,E1 14976.845,E2 14976.845} C_VEL
LIN {X 0,Y 374.745,Z 814.701,A -85,B 0,C 180,E1 14973.127,E2 14973.127} C_VEL
LIN {X 0,Y 374.187,Z 808.071,A -85,B 0,C 180,E1 14972.781,E2 14972.781} C_VEL
LIN {X 0,Y 366.246,Z 792.644,A -85,B 0,C 180,E1 14970.335,E2 14970.335} C_VEL
LIN {X 0,Y 358.54,Z 778.671,A -85,B 0,C 180,E1 14967.711,E2 14967.711} C_VEL
LIN {X 0,Y 351.584,Z 766.993,A -85,B 0,C 180,E1 14965.07,E2 14965.07} C_VEL
LIN {X 0,Y 346.438,Z 758.68,A -85,B 0,C 180,E1 14962.886,E2 14962.886} C_VEL
LIN {X 0,Y 341.091,Z 750.184,A -85,B 0,C 180,E1 14960.326,E2 14960.326} C_VEL
LIN {X 0,Y 336.499,Z 743.319,A -85,B 0,C 180,E1 14957.821,E2 14957.821} C_VEL
LIN {X 0,Y 334.366,Z 739.948,A -85,B 0,C 180,E1 14956.503,E2 14956.503} C_VEL
LIN {X 0,Y 330.963,Z 734.902,A -85,B 0,C 180,E1 14954.164,E2 14954.164} C_VEL
LIN {X 0,Y 327.878,Z 730.031,A -85,B 0,C 180,E1 14951.611,E2 14951.611} C_VEL
LIN {X 0,Y 325.298,Z 726.464,A -85,B 0,C 180,E1 14949.018,E2 14949.018} C_VEL
LIN {X 0,Y 324.607,Z 725.113,A -85,B 0,C 180,E1 14948.145,E2 14948.145} C_VEL
LIN {X 0,Y 320.677,Z 722.188,A -85,B 0,C 180,E1 14940,E2 14940} C_VEL
LIN {X 0,Y 320.869,Z 722.456,A -85,B 0,C 180,E1 14936.248,E2 14936.248} C_VEL
LIN {X 0,Y 324.891,Z 725.347,A -85,B 0,C 180,E1 14929,E2 14929} C_VEL
LIN {X 0,Y 326.898,Z 729.049,A -85,B 0,C 180,E1 14926.738,E2 14926.738} C_VEL
LIN {X 0,Y 330.205,Z 731.815,A -85,B 0,C 180,E1 14924.05,E2 14924.05} C_VEL
LIN {X 0,Y 332.907,Z 735.849,A -85,B 0,C 180,E1 14922.07,E2 14922.07} C_VEL
LIN {X 0,Y 335.269,Z 738.026,A -85,B 0,C 180,E1 14920.623,E2 14920.623} C_VEL
LIN {X 0,Y 338.448,Z 742.285,A -85,B 0,C 180,E1 14918.783,E2 14918.783} C_VEL
LIN {X 0,Y 340.151,Z 744.16,A -85,B 0,C 180,E1 14917.898,E2 14917.898} C_VEL
LIN {X 0,Y 343.893,Z 748.768,A -85,B 0,C 180,E1 14916.071,E2 14916.071} C_VEL
LIN {X 0,Y 349.267,Z 755.906,A -85,B 0,C 180,E1 14913.704,E2 14913.704} C_VEL
LIN {X 0,Y 353.744,Z 761.955,A -85,B 0,C 180,E1 14911.926,E2 14911.926} C_VEL
LIN {X 0,Y 361.999,Z 773.397,A -85,B 0,C 180,E1 14908.994,E2 14908.994} C_VEL
LIN {X 0,Y 371.283,Z 787.581,A -85,B 0,C 180,E1 14906.074,E2 14906.074} C_VEL
LIN {X 0,Y 374.728,Z 793.361,A -85,B 0,C 180,E1 14905.065,E2 14905.065} C_VEL
LIN {X 0,Y 365.742,Z 945.726,A -85,B 0,C 180,E1 14901.974,E2 14901.974} C_VEL
LIN {X 0,Y 363.897,Z 967.912,A -85,B 0,C 180,E1 14901.273,E2 14901.273} C_VEL
LIN {X 0,Y 361.176,Z 989.171,A -85,B 0,C 180,E1 14900.347,E2 14900.347} C_VEL
LIN {X 0,Y 357.735,Z 1008.692,A -85,B 0,C 180,E1 14899.237,E2 14899.237} C_VEL
LIN {X 0,Y 353.191,Z 1029.578,A -85,B 0,C 180,E1 14897.754,E2 14897.754} C_VEL
LIN {X 0,Y 348.52,Z 1047.681,A -85,B 0,C 180,E1 14896.178,E2 14896.178} C_VEL
LIN {X 0,Y 343.076,Z 1065.666,A -85,B 0,C 180,E1 14894.265,E2 14894.265} C_VEL
LIN {X 0,Y 337.057,Z 1083.426,A -85,B 0,C 180,E1 14891.983,E2 14891.983} C_VEL
LIN {X 0,Y 331.269,Z 1099.106,A -85,B 0,C 180,E1 14889.556,E2 14889.556} C_VEL
LIN {X 0,Y 325.377,Z 1113.761,A -85,B 0,C 180,E1 14886.813,E2 14886.813} C_VEL
LIN {X 0,Y 319.761,Z 1127.037,A -85,B 0,C 180,E1 14883.819,E2 14883.819} C_VEL
LIN {X 0,Y 314.482,Z 1139.235,A -85,B 0,C 180,E1 14880.501,E2 14880.501} C_VEL
LIN {X 0,Y 309.708,Z 1150.129,A -85,B 0,C 180,E1 14876.869,E2 14876.869} C_VEL
LIN {X 0,Y 305.796,Z 1159.201,A -85,B 0,C 180,E1 14873.101,E2 14873.101} C_VEL
LIN {X 0,Y 302.546,Z 1167.239,A -85,B 0,C 180,E1 14868.897,E2 14868.897} C_VEL
LIN {X 0,Y 300.397,Z 1173.206,A -85,B 0,C 180,E1 14864.85,E2 14864.85} C_VEL
LIN {X 0,Y 299.034,Z 1177.508,A -85,B 0,C 180,E1 14860.792,E2 14860.792} C_VEL
LIN {X 0,Y 298.234,Z 1180.511,A -85,B 0,C 180,E1 14856.545,E2 14856.545} C_VEL
LIN {X 0,Y 297.924,Z 1182.059,A -85,B 0,C 180,E1 14852.5,E2 14852.5} C_VEL
LIN {X 0,Y 297.883,Z 1182.168,A -85,B 0,C 180,E1 14848.461,E2 14848.461} C_VEL
LIN {X 0,Y 298.134,Z 1180.963,A -85,B 0,C 180,E1 14844.226,E2 14844.226} C_VEL
LIN {X 0,Y 298.799,Z 1178.442,A -85,B 0,C 180,E1 14840.174,E2 14840.174} C_VEL
LIN {X 0,Y 299.962,Z 1174.445,A -85,B 0,C 180,E1 14836.114,E2 14836.114} C_VEL
LIN {X 0,Y 301.925,Z 1168.986,A -85,B 0,C 180,E1 14832.063,E2 14832.063} C_VEL
LIN {X 0,Y 304.746,Z 1161.835,A -85,B 0,C 180,E1 14828.036,E2 14828.036} C_VEL
LIN {X 0,Y 308.347,Z 1153.255,A -85,B 0,C 180,E1 14824.246,E2 14824.246} C_VEL
LIN {X 0,Y 312.911,Z 1142.843,A -85,B 0,C 180,E1 14820.523,E2 14820.523} C_VEL
LIN {X 0,Y 317.848,Z 1131.654,A -85,B 0,C 180,E1 14817.245,E2 14817.245} C_VEL
LIN {X 0,Y 323.437,Z 1118.498,A -85,B 0,C 180,E1 14814.09,E2 14814.09} C_VEL
LIN {X 0,Y 327.093,Z 1109.666,A -85,B 0,C 180,E1 14812.268,E2 14812.268} C_VEL
LIN {X 0,Y 328.364,Z 1104.908,A -85,B 0,C 180,E1 14811.217,E2 14811.217} C_VEL
LIN {X 0,Y 328.879,Z 1093.134,A -85,B 0,C 180,E1 14808.374,E2 14808.374} C_VEL
LIN {X 0,Y 330.194,Z 1087.778,A -85,B 0,C 180,E1 14807.426,E2 14807.426} C_VEL
LIN {X 0,Y 336.19,Z 1071.189,A -85,B 0,C 180,E1 14805.184,E2 14805.184} C_VEL
LIN {X 0,Y 341.745,Z 1053.736,A -85,B 0,C 180,E1 14803.24,E2 14803.24} C_VEL
LIN {X 0,Y 347.061,Z 1034.779,A -85,B 0,C 180,E1 14801.495,E2 14801.495} C_VEL
LIN {X 0,Y 351.518,Z 1016.09,A -85,B 0,C 180,E1 14800.082,E2 14800.082} C_VEL
LIN {X 0,Y 355.268,Z 996.47,A -85,B 0,C 180,E1 14798.895,E2 14798.895} C_VEL
LIN {X 0,Y 358.417,Z 975.21,A -85,B 0,C 180,E1 14797.883,E2 14797.883} C_VEL
LIN {X 0,Y 360.502,Z 955.043,A -85,B 0,C 180,E1 14797.162,E2 14797.162} C_VEL
LIN {X 0,Y 362.241,Z 925.583,A -85,B 0,C 180,E1 14796.448,E2 14796.448} C_VEL
LIN {X 0,Y 370.075,Z 797.101,A -85,B 0,C 180,E1 14793.848,E2 14793.848} C_VEL
LIN {X 0,Y 361.199,Z 783.154,A -85,B 0,C 180,E1 14791.036,E2 14791.036} C_VEL
LIN {X 0,Y 352.888,Z 770.962,A -85,B 0,C 180,E1 14788.057,E2 14788.057} C_VEL
LIN {X 0,Y 345.447,Z 760.833,A -85,B 0,C 180,E1 14784.998,E2 14784.998} C_VEL
LIN {X 0,Y 341.211,Z 755.416,A -85,B 0,C 180,E1 14783.029,E2 14783.029} C_VEL
LIN {X 0,Y 337.343,Z 750.386,A -85,B 0,C 180,E1 14781.017,E2 14781.017} C_VEL
LIN {X 0,Y 333.831,Z 745.949,A -85,B 0,C 180,E1 14778.964,E2 14778.964} C_VEL
LIN {X 0,Y 332.789,Z 744.732,A -85,B 0,C 180,E1 14778.307,E2 14778.307} C_VEL
LIN {X 0,Y 329.62,Z 741.1,A -85,B 0,C 180,E1 14776.115,E2 14776.115} C_VEL
LIN {X 0,Y 328.481,Z 739.143,A -85,B 0,C 180,E1 14775.176,E2 14775.176} C_VEL
LIN {X 0,Y 325.156,Z 736.171,A -85,B 0,C 180,E1 14772.25,E2 14772.25} C_VEL
LIN {X 0,Y 323.609,Z 733.047,A -85,B 0,C 180,E1 14770.324,E2 14770.324} C_VEL
LIN {X 0,Y 319.903,Z 730.368,A -85,B 0,C 180,E1 14762.15,E2 14762.15} C_VEL
LIN {X 0,Y 320.399,Z 730.973,A -85,B 0,C 180,E1 14757.675,E2 14757.675} C_VEL
LIN {X 0,Y 323.747,Z 733.354,A -85,B 0,C 180,E1 14751.922,E2 14751.922} C_VEL
LIN {X 0,Y 325.946,Z 737.143,A -85,B 0,C 180,E1 14749.394,E2 14749.394} C_VEL
LIN {X 0,Y 327.059,Z 738.554,A -85,B 0,C 180,E1 14748.36,E2 14748.36} C_VEL
LIN {X 0,Y 330.644,Z 744.291,A -85,B 0,C 180,E1 14745.419,E2 14745.419} C_VEL
LIN {X 0,Y 333.908,Z 749.286,A -85,B 0,C 180,E1 14743.205,E2 14743.205} C_VEL
LIN {X 0,Y 337.63,Z 755.285,A -85,B 0,C 180,E1 14740.989,E2 14740.989} C_VEL
LIN {X 0,Y 341.964,Z 761.922,A -85,B 0,C 180,E1 14738.743,E2 14738.743} C_VEL
LIN {X 0,Y 348.365,Z 772.613,A -85,B 0,C 180,E1 14735.814,E2 14735.814} C_VEL
LIN {X 0,Y 354.787,Z 783.591,A -85,B 0,C 180,E1 14733.243,E2 14733.243} C_VEL
LIN {X 0,Y 362.451,Z 797.699,A -85,B 0,C 180,E1 14730.501,E2 14730.501} C_VEL
LIN {X 0,Y 370.089,Z 812.792,A -85,B 0,C 180,E1 14728.038,E2 14728.038} C_VEL
LIN {X 0,Y 370.2,Z 818.245,A -85,B 0,C 180,E1 14727.823,E2 14727.823} C_VEL
LIN {X 0,Y 357.652,Z 1026.173,A -85,B 0,C 180,E1 14723.608,E2 14723.608} C_VEL
LIN {X 0,Y 355.014,Z 1048.868,A -85,B 0,C 180,E1 14722.971,E2 14722.971} C_VEL
LIN {X 0,Y 351.137,Z 1071.057,A -85,B 0,C 180,E1 14722.154,E2 14722.154} C_VEL
LIN {X 0,Y 346.361,Z 1092.246,A -85,B 0,C 180,E1 14721.13,E2 14721.13} C_VEL
LIN {X 0,Y 341.179,Z 1111.794,A -85,B 0,C 180,E1 14719.895,E2 14719.895} C_VEL
LIN {X 0,Y 335.051,Z 1132.523,A -85,B 0,C 180,E1 14718.247,E2 14718.247} C_VEL
LIN {X 0,Y 328.83,Z 1151.651,A -85,B 0,C 180,E1 14716.357,E2 14716.357} C_VEL
LIN {X 0,Y 322.448,Z 1169.749,A -85,B 0,C 180,E1 14714.165,E2 14714.165} C_VEL
LIN {X 0,Y 315.915,Z 1187.686,A -85,B 0,C 180,E1 14711.532,E2 14711.532} C_VEL
LIN {X 0,Y 309.675,Z 1204.545,A -85,B 0,C 180,E1 14708.545,E2 14708.545} C_VEL
LIN {X 0,Y 304.163,Z 1219.431,A -85,B 0,C 180,E1 14705.348,E2 14705.348} C_VEL
LIN {X 0,Y 299.141,Z 1233.825,A -85,B 0,C 180,E1 14701.651,E2 14701.651} C_VEL
LIN {X 0,Y 295.253,Z 1246.168,A -85,B 0,C 180,E1 14697.86,E2 14697.86} C_VEL
LIN {X 0,Y 292.317,Z 1257.068,A -85,B 0,C 180,E1 14693.804,E2 14693.804} C_VEL
LIN {X 0,Y 290.468,Z 1266.094,A -85,B 0,C 180,E1 14689.714,E2 14689.714} C_VEL
LIN {X 0,Y 289.522,Z 1273.607,A -85,B 0,C 180,E1 14685.525,E2 14685.525} C_VEL
LIN {X 0,Y 289.319,Z 1279.007,A -85,B 0,C 180,E1 14681.562,E2 14681.562} C_VEL
LIN {X 0,Y 289.495,Z 1283.02,A -85,B 0,C 180,E1 14677.541,E2 14677.541} C_VEL
LIN {X 0,Y 289.791,Z 1285.148,A -85,B 0,C 180,E1 14673.957,E2 14673.957} C_VEL
LIN {X 0,Y 289.927,Z 1285.986,A -85,B 0,C 180,E1 14670.593,E2 14670.593} C_VEL
LIN {X 0,Y 289.847,Z 1285.548,A -85,B 0,C 180,E1 14667.034,E2 14667.034} C_VEL
LIN {X 0,Y 289.591,Z 1283.707,A -85,B 0,C 180,E1 14663.458,E2 14663.458} C_VEL
LIN {X 0,Y 289.323,Z 1280.202,A -85,B 0,C 180,E1 14659.446,E2 14659.446} C_VEL
LIN {X 0,Y 289.399,Z 1275.234,A -85,B 0,C 180,E1 14655.597,E2 14655.597} C_VEL
LIN {X 0,Y 290.159,Z 1268.095,A -85,B 0,C 180,E1 14651.309,E2 14651.309} C_VEL
LIN {X 0,Y 291.789,Z 1259.411,A -85,B 0,C 180,E1 14647.185,E2 14647.185} C_VEL
LIN {X 0,Y 294.418,Z 1249.006,A -85,B 0,C 180,E1 14643.15,E2 14643.15} C_VEL
LIN {X 0,Y 298.261,Z 1236.475,A -85,B 0,C 180,E1 14639.113,E2 14639.113} C_VEL
LIN {X 0,Y 303.016,Z 1222.68,A -85,B 0,C 180,E1 14635.422,E2 14635.422} C_VEL
LIN {X 0,Y 308.273,Z 1208.117,A -85,B 0,C 180,E1 14632.194,E2 14632.194} C_VEL
LIN {X 0,Y 314.712,Z 1190.839,A -85,B 0,C 180,E1 14629.001,E2 14629.001} C_VEL
LIN {X 0,Y 321.074,Z 1173.523,A -85,B 0,C 180,E1 14626.349,E2 14626.349} C_VEL
LIN {X 0,Y 327.574,Z 1155.132,A -85,B 0,C 180,E1 14624.045,E2 14624.045} C_VEL
LIN {X 0,Y 333.972,Z 1135.746,A -85,B 0,C 180,E1 14622.06,E2 14622.06} C_VEL
LIN {X 0,Y 340.035,Z 1115.744,A -85,B 0,C 180,E1 14620.399,E2 14620.399} C_VEL
LIN {X 0,Y 345.315,Z 1096.147,A -85,B 0,C 180,E1 14619.107,E2 14619.107} C_VEL
LIN {X 0,Y 350.275,Z 1074.775,A -85,B 0,C 180,E1 14618.018,E2 14618.018} C_VEL
LIN {X 0,Y 354.395,Z 1052.646,A -85,B 0,C 180,E1 14617.161,E2 14617.161} C_VEL
LIN {X 0,Y 357.247,Z 1030.08,A -85,B 0,C 180,E1 14616.493,E2 14616.493} C_VEL
LIN {X 0,Y 360.3,Z 981.996,A -85,B 0,C 180,E1 14615.483,E2 14615.483} C_VEL
LIN {X 0,Y 370.173,Z 815.845,A -85,B 0,C 180,E1 14612.119,E2 14612.119} C_VEL
LIN {X 0,Y 369.804,Z 812.305,A -85,B 0,C 180,E1 14611.909,E2 14611.909} C_VEL
LIN {X 0,Y 361.298,Z 795.569,A -85,B 0,C 180,E1 14609.147,E2 14609.147} C_VEL
LIN {X 0,Y 353.789,Z 781.963,A -85,B 0,C 180,E1 14606.43,E2 14606.43} C_VEL
LIN {X 0,Y 346.23,Z 769.051,A -85,B 0,C 180,E1 14603.32,E2 14603.32} C_VEL
LIN {X 0,Y 339.307,Z 757.736,A -85,B 0,C 180,E1 14599.988,E2 14599.988} C_VEL
LIN {X 0,Y 332.854,Z 747.641,A -85,B 0,C 180,E1 14596.222,E2 14596.222} C_VEL
LIN {X 0,Y 329.294,Z 742.313,A -85,B 0,C 180,E1 14593.7,E2 14593.7} C_VEL
LIN {X 0,Y 326.317,Z 737.549,A -85,B 0,C 180,E1 14591.13,E2 14591.13} C_VEL
LIN {X 0,Y 323.88,Z 733.843,A -85,B 0,C 180,E1 14588.521,E2 14588.521} C_VEL
LIN {X 0,Y 323.335,Z 732.926,A -85,B 0,C 180,E1 14587.82,E2 14587.82} C_VEL
LIN {X 0,Y 319.685,Z 730.103,A -85,B 0,C 180,E1 14579.82,E2 14579.82} C_VEL
LIN {X 0,Y 319.933,Z 730.467,A -85,B 0,C 180,E1 14576.057,E2 14576.057} C_VEL
LIN {X 0,Y 323.687,Z 733.256,A -85,B 0,C 180,E1 14569.229,E2 14569.229} C_VEL
LIN {X 0,Y 325.746,Z 736.962,A -85,B 0,C 180,E1 14566.871,E2 14566.871} C_VEL
LIN {X 0,Y 328.782,Z 739.614,A -85,B 0,C 180,E1 14564.342,E2 14564.342} C_VEL
LIN {X 0,Y 331.565,Z 743.672,A -85,B 0,C 180,E1 14562.267,E2 14562.267} C_VEL
LIN {X 0,Y 333.68,Z 745.753,A -85,B 0,C 180,E1 14560.936,E2 14560.936} C_VEL
LIN {X 0,Y 337.04,Z 750.129,A -85,B 0,C 180,E1 14558.964,E2 14558.964} C_VEL
LIN {X 0,Y 338.548,Z 752.029,A -85,B 0,C 180,E1 14558.153,E2 14558.153} C_VEL
LIN {X 0,Y 342.982,Z 757.746,A -85,B 0,C 180,E1 14555.958,E2 14555.958} C_VEL
LIN {X 0,Y 347.099,Z 763.189,A -85,B 0,C 180,E1 14554.124,E2 14554.124} C_VEL
LIN {X 0,Y 353.147,Z 771.438,A -85,B 0,C 180,E1 14551.699,E2 14551.699} C_VEL
LIN {X 0,Y 361.865,Z 784.174,A -85,B 0,C 180,E1 14548.611,E2 14548.611} C_VEL
LIN {X 0,Y 370.089,Z 797.342,A -85,B 0,C 180,E1 14546.019,E2 14546.019} C_VEL
LIN {X 0,Y 360.961,Z 946.616,A -85,B 0,C 180,E1 14542.976,E2 14542.976} C_VEL
LIN {X 0,Y 359.121,Z 968.424,A -85,B 0,C 180,E1 14542.29,E2 14542.29} C_VEL
LIN {X 0,Y 356.344,Z 989.518,A -85,B 0,C 180,E1 14541.374,E2 14541.374} C_VEL
